(* Logix 5000 project; controller Close_Palletizing 1769-L33ERM rev 33.13; software revision 33.00; part 4 of 5 *)

VAR_GLOBAL   (* controller tags *)
   ActiveUserFrame : DINT := 1;
   ActiveUserFrame_Old : DINT := 1;
   ActiveUserFrame_Timer : TIMER := (PRE := 50, ACC := 21, EN := 1, TT := 1);
   ActiveUserFrameErr : BOOL;
   AirPressure : ALIAS FOR YRC1000_Rbt_Ctlr:I.Data[1].4;   // Sensor on air in, used to verify pressure
   Alarm : ALIAS FOR YRC1000_Rbt_Ctlr:I.Data[8].3;   // Robot in Alarm state
   AlarmReset : ALIAS FOR YRC1000_Rbt_Ctlr:O.Data[0].3;   // Reset alarm output
   AtHomePosition : ALIAS FOR YRC1000_Rbt_Ctlr:I.Data[5].2;
   BatteryAlarm : ALIAS FOR YRC1000_Rbt_Ctlr:I.Data[8].4;   // Robot battery is low
   Blue1 : BOOL;
   Blue2 : BOOL;
   BoltBucketSensor : ALIAS FOR YRC1000_Rbt_Ctlr:I.Data[1].7;   // Sense if the Bolt Bucket is present in the stand
   BothPalletsEmpty : ALIAS FOR Palletizer_full_produced.1;
   BothPalletsFull : ALIAS FOR Palletizer_full_produced.2;
   CallMaster : ALIAS FOR YRC1000_Rbt_Ctlr:O.Data[0].2;   // Call master program to move pointer to top of Master Job
   CallMaster_Timer : TIMER := (PRE := 1000);
   cc_ONS1 : BOOL;
   cc_State : DINT := 100;
   CenterDist : DINT := 303000;
   CheckClearPallet : ALIAS FOR YRC1000_Rbt_Ctlr:I.Data[10].1;
   CheckForComplete : ALIAS FOR YRC1000_Rbt_Ctlr:I.Data[9].5;
   CheckForCompleteAcknowledge : ALIAS FOR YRC1000_Rbt_Ctlr:O.Data[4].6;
   ClearPalletAcknowledge : ALIAS FOR YRC1000_Rbt_Ctlr:O.Data[6].4;
   CloseOffset : DINT := 18;
   Conv_Seq : DINT;
   Conv_Seq_ONS : BOOL := 1;
   ConvConversion2 : REAL := 0.2444492;
   ConveyorActuatorExtend : BOOL;
   ConveyorActuatorRetract : BOOL := 1;
   ConveyorApproachLocation : YRC1000_POSITION_VAR := (Data_Type := 19, Tool_Num := 2, User_Coord_Num := 3, Axis1_Data := -45828, Axis2_Data := 300000, Axis3_Data := 145000, Axis4_Data := 1800000, Axis5_Data := 20000, Axis6_Data := 1800000);
   ConveyorHeight : REAL := 406.29633;   // Distance from UF 3 to the top of the conveyor
   ConveyorPickLocation : YRC1000_POSITION_VAR := (Data_Type := 19, Tool_Num := 2, User_Coord_Num := 3, Axis1_Data := -45828, Axis2_Data := 355000, Axis3_Data := 81500, Axis4_Data := 1800000, Axis5_Data := 20000, Axis6_Data := 1800000);
   ConveyorSequenceReset_Timer : TIMER := (PRE := 3000, ACC := 3000, EN := 1, DN := 1);
   ConveyorSpeed : REAL := 9.301;   // Speed of the conveyor in ft/min
   ConvMul1 : REAL := 1.0;
   ConvMul2 : REAL := 0.99;
   ConvMul3 : REAL := 1.01;
   CurrentPos : REAL[6] := ([0] := 900.002, [1] := 0.001, [2] := 600.006, [3] := -179.9997, [4] := -0.0009, [5] := -0.0009);   // Current position of the active TCP on the robot
   CurrentPos_micro : YRC1000_POSITION_VAR := (Data_Type := 16, Config := 16, Tool_Num := 1, Axis1_Data := 900002, Axis2_Data := 1, Axis3_Data := 600006, Axis4_Data := -1799997, Axis5_Data := -9, Axis6_Data := -9);   // μm
   currentPosErr : BOOL;
   CurrPos_Timer : TIMER := (PRE := 10);
   delay_GoToPick : TIMER := (PRE := 1000);
   delay_LeftPalletOff : TIMER := (PRE := 1000);
   delay_LeftPalletOn : TIMER := (PRE := 1000, ACC := 1000, EN := 1, DN := 1);
   delay_RightPalletOff : TIMER := (PRE := 1000);
   delay_RightPalletOn : TIMER := (PRE := 1000, ACC := 1000, EN := 1, DN := 1);
   DistanceInArray : INT[16] := ([0] := 1976);
        [0]   // Distance sensor reading in MM
   DistanceOutArray : INT[16];
   DistanceSensorValue : DINT := 1978000;
   DoorAccessRequested : ALIAS FOR YRC1000_Rbt_Ctlr:O.Data[5].3;
   DoorLatchRelayPower : ALIAS FOR YRC1000_Rbt_Ctlr:O.Data[2].2;   // Powers the relay that enables the door latch
   DoorRequestAccess : ALIAS FOR YRC1000_Rbt_Ctlr:I.Data[1].0;   // Door Interlock, For request Entry
   DoorUnlocked : ALIAS FOR YRC1000_Rbt_Ctlr:I.Data[2].0;   // The Door Latch is unlocked
   Error_RobotPickupFailed : ALIAS FOR YRC1000_Rbt_Ctlr:I.Data[9].3;
   ExtendedPartWidth : DINT := 693;
   ExtendGripper : ALIAS FOR YRC1000_Rbt_Ctlr:I.Data[9].0;
   ExternalHold : ALIAS FOR YRC1000_Rbt_Ctlr:O.Data[0].1;   // Pauses program execution
   ExternalStart : ALIAS FOR YRC1000_Rbt_Ctlr:O.Data[0].0;   // External command to start the program
   ExtServoOn : ALIAS FOR YRC1000_Rbt_Ctlr:O.Data[0].4;   // External command to turn servos on
   FanucLongPart : DINT := 1072;
   FanucMediumPart : DINT := 795;
   FanucShortPart : DINT := 465;
   GoToPartChange : ALIAS FOR YRC1000_Rbt_Ctlr:O.Data[6].0;
   GoToPick : ALIAS FOR YRC1000_Rbt_Ctlr:O.Data[6].1;
   Green1 : BOOL := 1;
   Green2 : BOOL;
   GrippedPartDistance : DINT := 46000;
   GrippedPartLatchDelay : TIMER := (PRE := 3000);
   HMI_HoldFanuc : BOOL;
   HMI_Manual : BOOL;
   HMI_ParkFanuc : BOOL;
   HMI_Reset : BOOL;
   HMI_Reset_Timer : TIMER := (PRE := 5000);
   HMI_ResetFanuc : BOOL;
   HMI_Start : BOOL;
   HMI_Start_Timer : TIMER := (PRE := 5000);
   HMI_StartFanuc : BOOL;
   HMI_Stop : ALIAS FOR YRC1000_Rbt_Ctlr:O.Data[5].4;
   IFM_Port1_Stroke : Generic_4PORT_IOL := (IOL_Mode := 1, Port_Process_Data_Size := 4, Port_Number := 1, Vendor_ID := 26, Device_ID := 8388785);   // Stroke sensor reading can be found in StrokeInputArray[0]
   IFM_Port2_Distance : Generic_4PORT_IOL := (IOL_Mode := 1, Port_Process_Data_Size := 4, Port_Number := 2, Vendor_ID := 26, Device_ID := 6488065);   // Distance sensor reading can be found in DistanceInArray[0]
   InchesToMove : DINT := 45;
   InHomePosition : ALIAS FOR YRC1000_Rbt_Ctlr:O.Data[5].7;
   InPartChange : ALIAS FOR YRC1000_Rbt_Ctlr:I.Data[9].7;
   InPickApproachAcknowledge : ALIAS FOR YRC1000_Rbt_Ctlr:O.Data[5].2;
   InPlay : ALIAS FOR YRC1000_Rbt_Ctlr:I.Data[8].6;   // Robot is in play mode
   InRemote : ALIAS FOR YRC1000_Rbt_Ctlr:I.Data[8].5;   // Robot is in remote mode
   InTeach : ALIAS FOR YRC1000_Rbt_Ctlr:I.Data[8].7;   // Robot is in teach mode
   LayerNum : DINT := 3;
   LayerPosition : DINT;
   LeftFlashOff : TIMER := (PRE := 750);
   LeftFlashOn : TIMER := (PRE := 750);
   LeftFullRightEmpty : ALIAS FOR Palletizer_full_produced.3;
   LeftIndicator_Green : ALIAS FOR YRC1000_Rbt_Ctlr:O.Data[1].6;   // Indicator light showing the pallet is complete
   LeftIndicator_Yellow : ALIAS FOR YRC1000_Rbt_Ctlr:O.Data[1].7;   // Indicator light showing the pallet is in progress / present
   LeftPalletComplete : ALIAS FOR YRC1000_Rbt_Ctlr:O.Data[4].0;
   LeftPalletPresent : ALIAS FOR YRC1000_Rbt_Ctlr:O.Data[6].6;
   LeftPalletSensor : ALIAS FOR YRC1000_Rbt_Ctlr:I.Data[1].2;   // Sense if a pallet is in the pallet holder
   LeftPalletWillBeNew : BOOL;
   msg_Read_ActiveUserFrame : MESSAGE;
        MessageParameters(ServiceCode := 16#000e, DestinationTag := ActiveUserFrame, ...)
   msg_Read_CurrentPosition : MESSAGE;   // Reading the current position of the robot
        MessageParameters(ServiceCode := 16#0001, DestinationTag := CurrentPos_micro, ...)
   msg_Read_PalletCount : MESSAGE;
        MessageParameters(ServiceCode := 16#000e, DestinationTag := PalletCount, ...)
   msg_Read_PartCount : MESSAGE;   // Reading Part Count from the robot
        MessageParameters(ServiceCode := 16#000e, DestinationTag := PartCount, ...)
   msg_Write_ActiveUserFrame : MESSAGE;
        MessageParameters(ServiceCode := 16#0010, LocalElement := ActiveUserFrame, ...)
   msg_Write_ConveyorApproachLocation : MESSAGE;
        MessageParameters(ServiceCode := 16#0010, LocalElement := ConveyorApproachLocation, ...)
   msg_Write_ConveyorPickLocation : MESSAGE;
        MessageParameters(ServiceCode := 16#0010, LocalElement := ConveyorPickLocation, ...)
   msg_Write_PalletCount : MESSAGE;
        MessageParameters(ServiceCode := 16#0010, LocalElement := PalletCount, ...)
   msg_Write_PalletPlaceLocation : MESSAGE;
        MessageParameters(ServiceCode := 16#0010, LocalElement := RadiatorPlaceLocation, ...)
   msg_Write_PartCount : MESSAGE;
        MessageParameters(ServiceCode := 16#0010, LocalElement := PartCount, ...)
   msg_Write_RadiatorType : MESSAGE;
        MessageParameters(ServiceCode := 16#0010, LocalElement := RadiatorType, ...)
   NewPallet : ALIAS FOR YRC1000_Rbt_Ctlr:O.Data[6].3;
   OffsetDist : DINT := 214000;
   ONS_PartGripped : BOOL;
   ons_SendFanucHome : BOOL;
   ons_StartClearPallet : BOOL;
   PalletCount : DINT := 5;
   PalletCount_old : DINT := 4;
   PalletCount_Timer : TIMER := (PRE := 50, ACC := 9, EN := 1, TT := 1);
   PalletCountErr : BOOL;
   Palletizer_full_produced : DINT := 46596096; {produced}
   PalletNotClear : ALIAS FOR YRC1000_Rbt_Ctlr:O.Data[6].5;
   PalletsNotReady : BOOL;
   PalletStarted : ALIAS FOR YRC1000_Rbt_Ctlr:I.Data[10].2;
   PartCount : DINT := 5;
   PartCount_Timer : TIMER := (PRE := 50, ACC := 10, EN := 1, TT := 1);
   PartCountErr : BOOL;
   PartID_Current : DINT := 7;
   PartInTool : ALIAS FOR YRC1000_Rbt_Ctlr:O.Data[4].2;
   PartLength : DINT := 432;
   PartLength_Current : DINT := 432;   // 17" = 432 mm | 30" = 762 mm | 41" = 1041 mm
   PartMovedOn_Timer : TIMER := (PRE := 14667);
   PartNeverReachedEnd : ALIAS FOR Palletizer_full_produced.6;
   PartNeverReachedEnd_Timer : TIMER := (PRE := 24191);
   PartNum : DINT := 5990261;
   PartNum_Current : DINT := 5990261;
   PartNumber : STRING := '5990261L';
   PartNumber_Current : STRING := '5990261L';
   PartPosition : DINT;
   PartRows : DINT := 3;
   PartRows_Current : DINT := 3;
   PartThickness : REAL := 51.5;
   PartThickness_Current : REAL := 51.5;   // 2r = 34.1-34.6 mm | 3r = 51.1-51.8 mm | 4r = 68.2-68.9 mm
   PartWidth : DINT := 711;
   PartWidth_Current : DINT := 711;   // 14" = 356 mm | 16" = 407 mm | 20" = 508 mm | 22" = 559 mm | 24" = 610 mm | 28" = 711 mm | 32" = 813 mm
   PCConnect : STRING := '1/24/2024 3:13:43 PM';
   Pick_Seq : DINT;
   Pick_Timer : TIMER := (PRE := 1000);
   PickConversion1 : REAL := 3.75;
   PickConversion2 : REAL := 225000.0;
   PickReq_State : DINT := 10;
   PickRequest : ALIAS FOR YRC1000_Rbt_Ctlr:I.Data[9].6;
   PickRequestAcknowledge : ALIAS FOR YRC1000_Rbt_Ctlr:O.Data[5].5;
   PickupConveyorSensor : ALIAS FOR YRC1000_Rbt_Ctlr:I.Data[1].5;   // Sense if the radiator is ready for pickup
   PickupErrorAcknowledge : ALIAS FOR YRC1000_Rbt_Ctlr:O.Data[4].7;
   pickupRecovery : BOOL;
   PickupSensorInactive_Timer : TIMER := (PRE := 5000);
   Place_Error : BOOL;
   PlaceReq_State : DINT := 10;
   PlaceRequestAcknowledge : ALIAS FOR YRC1000_Rbt_Ctlr:O.Data[4].5;
   PN_Timer : TIMER := (PRE := 10);
   Prog_StartFanuc : BOOL;
   QuadStack : ALIAS FOR YRC1000_Rbt_Ctlr:O.Data[5].1;
   RadiatorPicked : ALIAS FOR Palletizer_full_produced.0;
   RadiatorPlaceLocation : YRC1000_POSITION_VAR := (Data_Type := 19, Tool_Num := 8, User_Coord_Num := 1, Axis1_Data := 517000, Axis3_Data := 316750, Axis4_Data := 1800000);
   RadiatorType : DINT := 1;   // 1: 17" 2: 30" 3 41"
   Read_ActiveUserFrame : BOOL;
   Read_CurrPos : BOOL := 1;
   Read_PalletCount : BOOL;
   Read_PartCount : BOOL := 1;
   Release_Timer : TIMER := (PRE := 5000);
   Reset : ALIAS FOR YRC1000_Rbt_Ctlr:I.Data[1].1;   // Door Interlock, For reset Entry
   ResetPalletCount : BOOL;
   RetractGripper : ALIAS FOR YRC1000_Rbt_Ctlr:I.Data[9].1;
   RightFlashOff : TIMER := (PRE := 750, ACC := 174, EN := 1, TT := 1);
   RightFlashOn : TIMER := (PRE := 750, ACC := 750, EN := 1, DN := 1);
   RightFullLeftEmpty : ALIAS FOR Palletizer_full_produced.4;
   RightIndicator_Green : ALIAS FOR YRC1000_Rbt_Ctlr:O.Data[2].0;   // Indicator light showing the pallet is complete
   RightIndicator_Yellow : ALIAS FOR YRC1000_Rbt_Ctlr:O.Data[2].1;   // Indicator light showing the pallet is in progress / present
   RightPalletComplete : ALIAS FOR YRC1000_Rbt_Ctlr:O.Data[4].1;
   RightPalletPresent : ALIAS FOR YRC1000_Rbt_Ctlr:O.Data[6].7;
   RightPalletSensor : ALIAS FOR YRC1000_Rbt_Ctlr:I.Data[1].3;   // Sense if a pallet is in the pallet holder
   RightPalletWillBeNew : BOOL;
   Robot_InPickApproach : ALIAS FOR YRC1000_Rbt_Ctlr:I.Data[9].4;
   RobotCannotPlaceCurrentPart : ALIAS FOR Palletizer_full_produced.5;
   RobotExternalEStop : ALIAS FOR YRC1000_Rbt_Ctlr:I.Data[4].1;
   RobotInsideConveyor : ALIAS FOR YRC1000_Rbt_Ctlr:I.Data[10].0;
   RobotInsideConveyorProduced : ALIAS FOR Palletizer_full_produced.9;
   RobotNotRunning : ALIAS FOR Palletizer_full_produced.7;
   RobotNotSupposedToBeRunning : ALIAS FOR Palletizer_full_produced.8;
   RobotPlaceRequest : ALIAS FOR YRC1000_Rbt_Ctlr:I.Data[9].2;
   RobotTeachPendantEStop : ALIAS FOR YRC1000_Rbt_Ctlr:I.Data[4].2;
   Running : ALIAS FOR YRC1000_Rbt_Ctlr:I.Data[8].0;   // Robot running status
   SafetyCircuitBroken : ALIAS FOR YRC1000_Rbt_Ctlr:I.Data[4].0;
   SafetyRelayReset : ALIAS FOR YRC1000_Rbt_Ctlr:O.Data[2].3;   // Reset the safety relays linked to the Pilz sensors
   SecondConveyorSensor : ALIAS FOR YRC1000_Rbt_Ctlr:I.Data[1].6;   // Sense if a coil is waiting on the conveyor
   SelectPlay : ALIAS FOR YRC1000_Rbt_Ctlr:O.Data[0].5;   // External command to put robot in play mode
   SelectTeach : ALIAS FOR YRC1000_Rbt_Ctlr:O.Data[0].6;   // External command to put robot in teach mode
   ServoOn : ALIAS FOR YRC1000_Rbt_Ctlr:I.Data[8].1;   // Servo on status
   SideDist : DINT;
   SingleStack : ALIAS FOR YRC1000_Rbt_Ctlr:O.Data[5].0;
   StackLight_Blue : ALIAS FOR YRC1000_Rbt_Ctlr:O.Data[1].3;   // Blue on the light stack
   StackLight_Buzzer : ALIAS FOR YRC1000_Rbt_Ctlr:O.Data[1].0;   // Buzzer on the stack light
   StackLight_Green : ALIAS FOR YRC1000_Rbt_Ctlr:O.Data[1].5;   // Green light on light stack
   StackLight_Red : ALIAS FOR YRC1000_Rbt_Ctlr:O.Data[1].2;   // Red light on light stack
   StackLight_White : ALIAS FOR YRC1000_Rbt_Ctlr:O.Data[1].1;   // White on the light stack
   StackLight_Yellow : ALIAS FOR YRC1000_Rbt_Ctlr:O.Data[1].4;   // Yellow light on light stack
   state_CheckClearPallet : DINT := 100;
   StillOnOldPart_Timer : TIMER := (PRE := 500);
   StrokeInputArray : INT[16] := ([0] := 13136);
   StrokeOutputArray : INT[16];
   StrokePosition : DINT := 821;   // Gripper Cylinder position GTE 700 = Retracted LTE 100 = Extended
   test_bit_1 : BOOL := 1;
   test_bit_2 : BOOL;
   test_bit_3 : BOOL := 1;
   test_toggle : BOOL;
   ThirdConveyorSensor : BOOL;
   timer_FanucReset : TIMER := (PRE := 500);
   timer_FanucStart : TIMER := (PRE := 500);
   timer_GreenFlashOff : TIMER := (PRE := 1000, ACC := 1000, EN := 1, DN := 1);
   timer_GreenFlashOn : TIMER := (PRE := 1000, ACC := 351, EN := 1, TT := 1);
   ToolExtended : ALIAS FOR YRC1000_Rbt_Ctlr:O.Data[4].3;
   ToolRetracted : ALIAS FOR YRC1000_Rbt_Ctlr:O.Data[4].4;
   ToPC_AirPressure : DINT := 1;
   ToPC_BoltBucketSensor : DINT := 1;
   ToPC_ConveyorStatus : DINT;
   ToPC_DoorStatus : DINT;
   ToPC_FanucFault : DINT := 1;
   ToPC_FanucRunning : DINT;
   ToPC_LeftPalletStatus : DINT := 1;
   ToPC_PalletNotClear : DINT;
   ToPC_PickupFailed : DINT;
   ToPC_PlaceError : DINT;
   ToPC_RightPalletStatus : DINT := 2;
   ToPC_RobotEStop : DINT;
   ToPC_RobotRunning : DINT := 1;
   ToPC_SafetyCircuitBroken : DINT;
   ToPC_ToolStatus : DINT;
   TopOfMaster : ALIAS FOR YRC1000_Rbt_Ctlr:I.Data[8].2;   // Top of Master Job
   TurnOffBuzzer : BOOL;
   TwoStack : ALIAS FOR YRC1000_Rbt_Ctlr:O.Data[6].2;
   WaitingForPartAtEnd : BOOL;
   Write_ActiveUserFrame : BOOL;
   Write_ActiveUserFrame1 : BOOL;
   Write_ConveyorLocations : BOOL;
   Write_PalletPlaceLocation : BOOL;
   Write_PartCount : BOOL;
   Write_RadiatorType : BOOL;
END_VAR

PROGRAM MainProgram   (* main routine MainRoutine *)
VAR
   ActuatorCloseTime : REAL := 0.75;
   ConvConversion : REAL := 74.50812;
   ConvConversion1 : REAL := 6.2090096;
   ConveyorLocations_ONS : BOOL;
   ConvMultiplier : REAL := 1.0;
   ToggleStokeAOI : BOOL := 1;
   Write_ActiveUserFrame2 : BOOL;
END_VAR

ROUTINE Fanuc_Communication   (* ladder *)
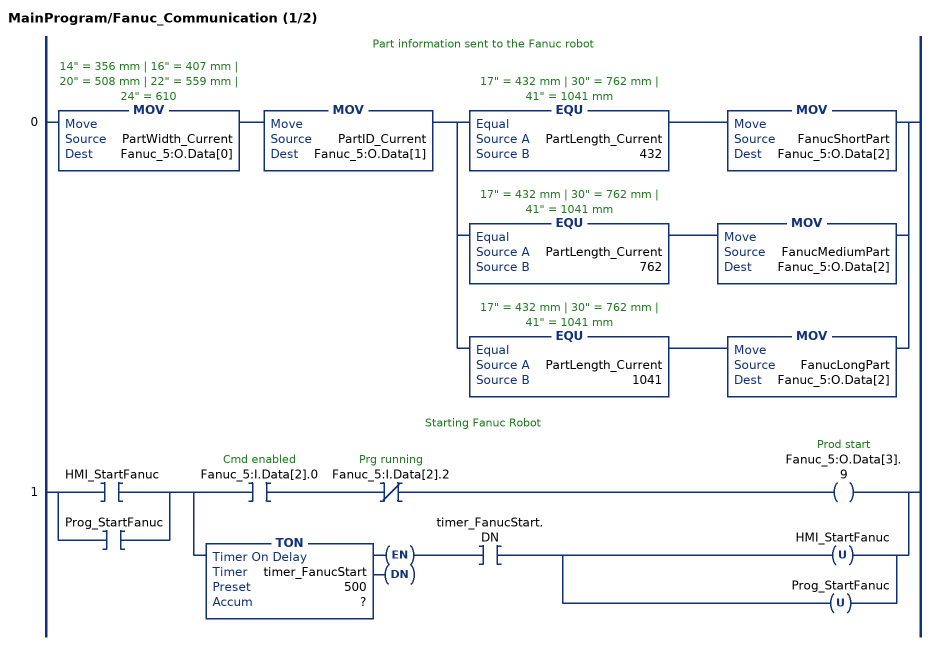
   // Part information sent to the Fanuc robot
   0: MOV(PartWidth_Current,Fanuc_5:O.Data[0])MOV(PartID_Current,Fanuc_5:O.Data[1])[EQU(PartLength_Current,432) MOV(FanucShortPart,Fanuc_5:O.Data[2]) ,EQU(PartLength_Current,762) MOV(FanucMediumPart,Fanuc_5:O.Data[2]) ,EQU(PartLength_Current,1041) MOV(FanucLongPart,Fanuc_5:O.Data[2]) ];
   // Starting Fanuc Robot
   1: [XIC(HMI_StartFanuc) ,XIC(Prog_StartFanuc) ][XIC(Fanuc_5:I.Data[2].0) XIO(Fanuc_5:I.Data[2].2) OTE(Fanuc_5:O.Data[3].9) ,TON(timer_FanucStart,?,?) XIC(timer_FanucStart.DN) [OTU(HMI_StartFanuc) ,OTU(Prog_StartFanuc) ] ];
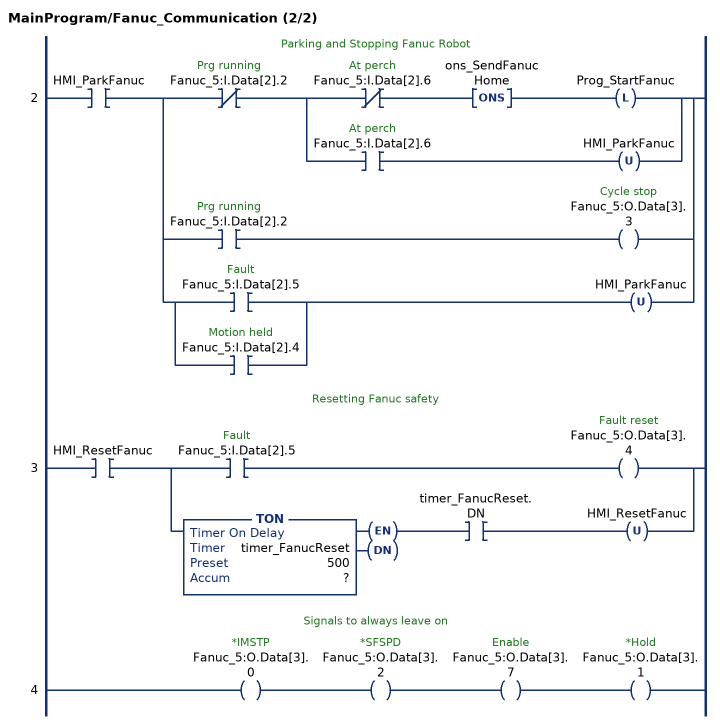
   // Parking and Stopping Fanuc Robot
   2: XIC(HMI_ParkFanuc)[[XIO(Fanuc_5:I.Data[2].2) [XIO(Fanuc_5:I.Data[2].6) ONS(ons_SendFanucHome) OTL(Prog_StartFanuc) ,XIC(Fanuc_5:I.Data[2].6) OTU(HMI_ParkFanuc) ] ,XIC(Fanuc_5:I.Data[2].2) OTE(Fanuc_5:O.Data[3].3) ] ,[XIC(Fanuc_5:I.Data[2].5) ,XIC(Fanuc_5:I.Data[2].4) ] OTU(HMI_ParkFanuc) ];
   // Resetting Fanuc safety
   3: XIC(HMI_ResetFanuc)[XIC(Fanuc_5:I.Data[2].5) OTE(Fanuc_5:O.Data[3].4) ,TON(timer_FanucReset,?,?) XIC(timer_FanucReset.DN) OTU(HMI_ResetFanuc) ];
   // Signals to always leave on
   4: OTE(Fanuc_5:O.Data[3].0)OTE(Fanuc_5:O.Data[3].2)OTE(Fanuc_5:O.Data[3].7)OTE(Fanuc_5:O.Data[3].1);
END_ROUTINE

ROUTINE Fanuc_PartID   (* structured text *)
   if PartLength_Current = 432 then
   	if PartWidth_Current = 356 then
   		PartID_Current := 1;
   	elsif PartWidth_Current = 406 then
   		PartID_Current := 2;
   	elsif PartWidth_Current = 508 then
   		if PartRows_Current = 2 then
   			PartID_Current := 3;
   		elsif PartRows_Current = 3 then
   			PartID_Current := 4;
   		end_if;
   	elsif PartWidth_Current = 559 then
   		PartID_Current := 5;
   	elsif PartWidth_Current = 610 then
   		PartID_Current := 6;
   	elsif PartWidth_Current = 711 then
   		if PartRows_Current = 3 then
   			PartID_Current := 7;
   		elsif PartRows_Current = 4 then
   			PartID_Current := 8;
   		end_if;
   	elsif PartWidth_Current = 813 then
   		PartID_Current := 9;
   	end_if;
   elsif PartLength_Current = 762 then
   	if PartRows_Current = 2 then
   		PartID_Current := 10;
   	elsif PartRows_Current = 3 then
   		PartID_Current := 11;
   	end_if;
   elsif PartLength_Current = 1041 then
   	if PartRows_Current = 3 then
   		PartID_Current := 12;
   	elsif PartRows_Current = 4 then
   		PartID_Current := 13;
   	end_if;
   end_if;
END_ROUTINE

ROUTINE IO_Link   (* ladder *)
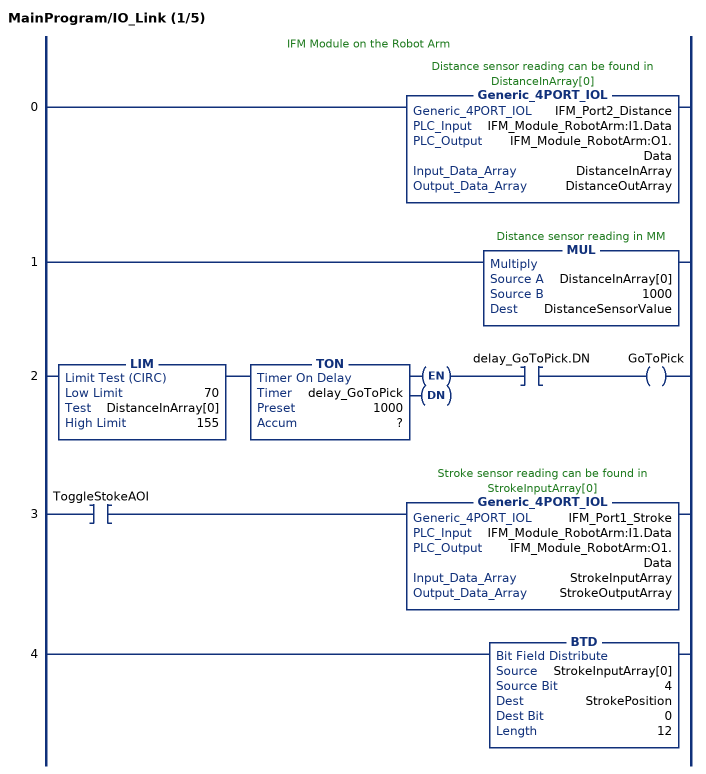
   // IFM Module on the Robot Arm
   0: Generic_4PORT_IOL(IFM_Port2_Distance,IFM_Module_RobotArm:I1.Data,IFM_Module_RobotArm:O1.Data,DistanceInArray,DistanceOutArray);
   1: MUL(DistanceInArray[0],1000,DistanceSensorValue);
   2: LIM(70,DistanceInArray[0],155)TON(delay_GoToPick,?,?)XIC(delay_GoToPick.DN)OTE(GoToPick);
   3: XIC(ToggleStokeAOI)Generic_4PORT_IOL(IFM_Port1_Stroke,IFM_Module_RobotArm:I1.Data,IFM_Module_RobotArm:O1.Data,StrokeInputArray,StrokeOutputArray);
   4: BTD(StrokeInputArray[0],4,StrokePosition,0,12);
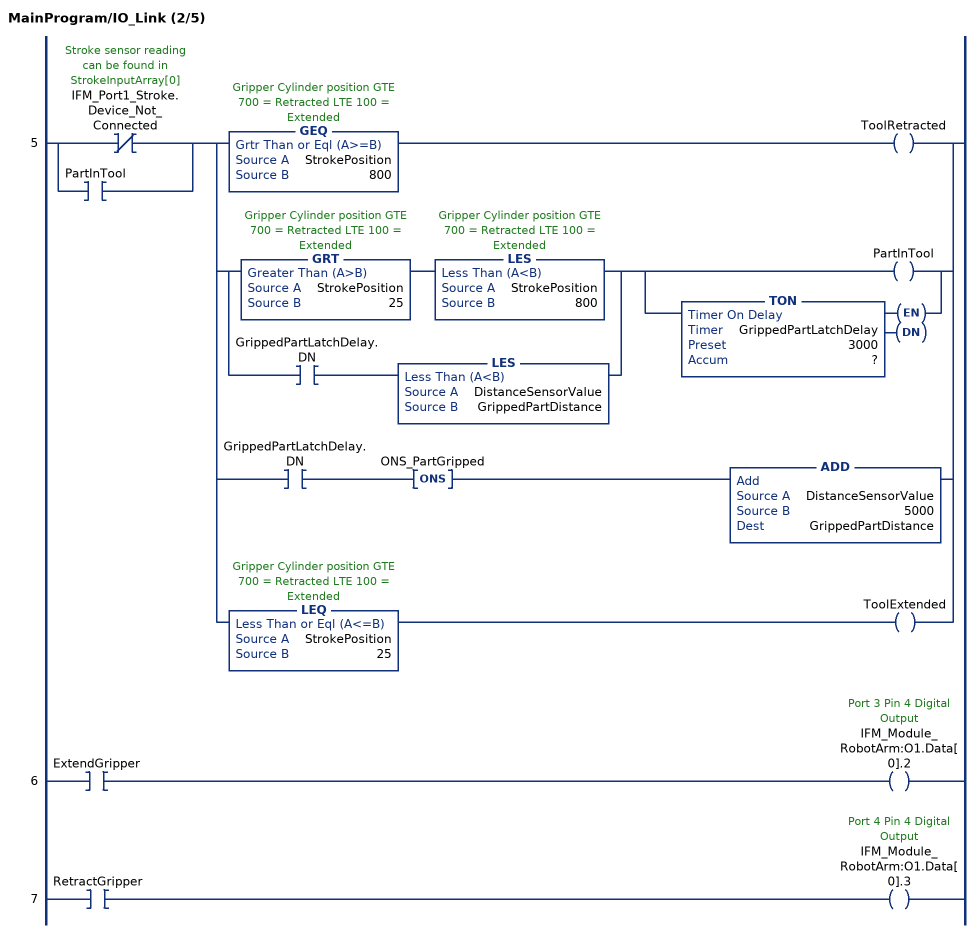
   5: [XIO(IFM_Port1_Stroke.Device_Not_Connected) ,XIC(PartInTool) ][GEQ(StrokePosition,800) OTE(ToolRetracted) ,[GRT(StrokePosition,25) LES(StrokePosition,800) ,XIC(GrippedPartLatchDelay.DN) LES(DistanceSensorValue,GrippedPartDistance) ] [OTE(PartInTool) ,TON(GrippedPartLatchDelay,?,?) ] ,XIC(GrippedPartLatchDelay.DN) ONS(ONS_PartGripped) ADD(DistanceSensorValue,5000,GrippedPartDistance) ,LEQ(StrokePosition,25) OTE(ToolExtended) ];
   6: XIC(ExtendGripper)OTE(IFM_Module_RobotArm:O1.Data[0].2);
   7: XIC(RetractGripper)OTE(IFM_Module_RobotArm:O1.Data[0].3);
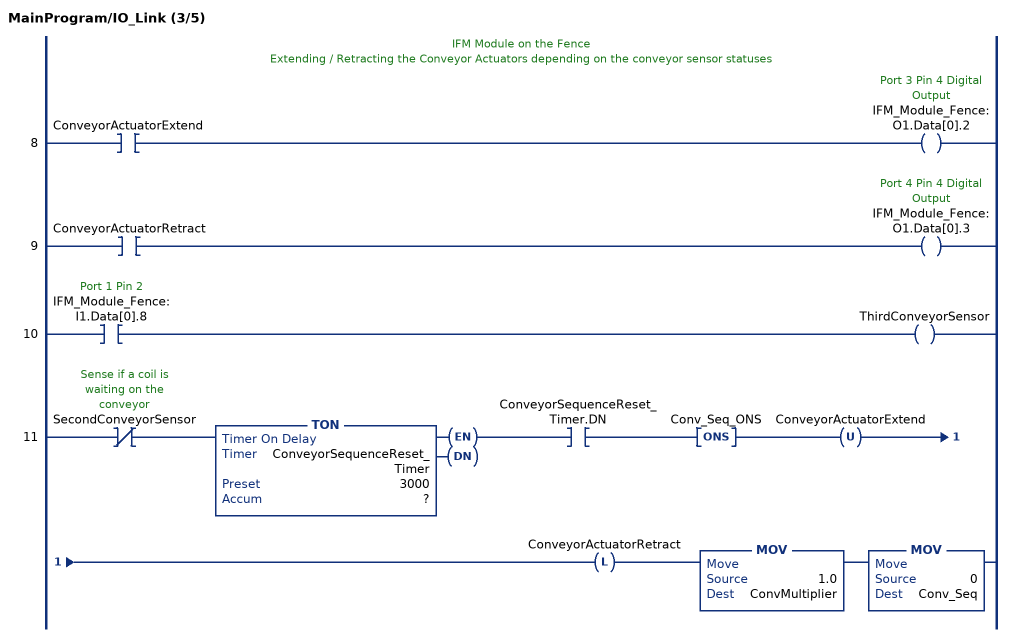
   // IFM Module on the Fence
   // Extending / Retracting the Conveyor Actuators depending on the conveyor sensor statuses
   8: XIC(ConveyorActuatorExtend)OTE(IFM_Module_Fence:O1.Data[0].2);
   9: XIC(ConveyorActuatorRetract)OTE(IFM_Module_Fence:O1.Data[0].3);
   10: XIC(IFM_Module_Fence:I1.Data[0].8)OTE(ThirdConveyorSensor);
   11: XIO(SecondConveyorSensor)TON(ConveyorSequenceReset_Timer,?,?)XIC(ConveyorSequenceReset_Timer.DN)ONS(Conv_Seq_ONS)OTU(ConveyorActuatorExtend)OTL(ConveyorActuatorRetract)MOV(1.0,ConvMultiplier)MOV(0,Conv_Seq);
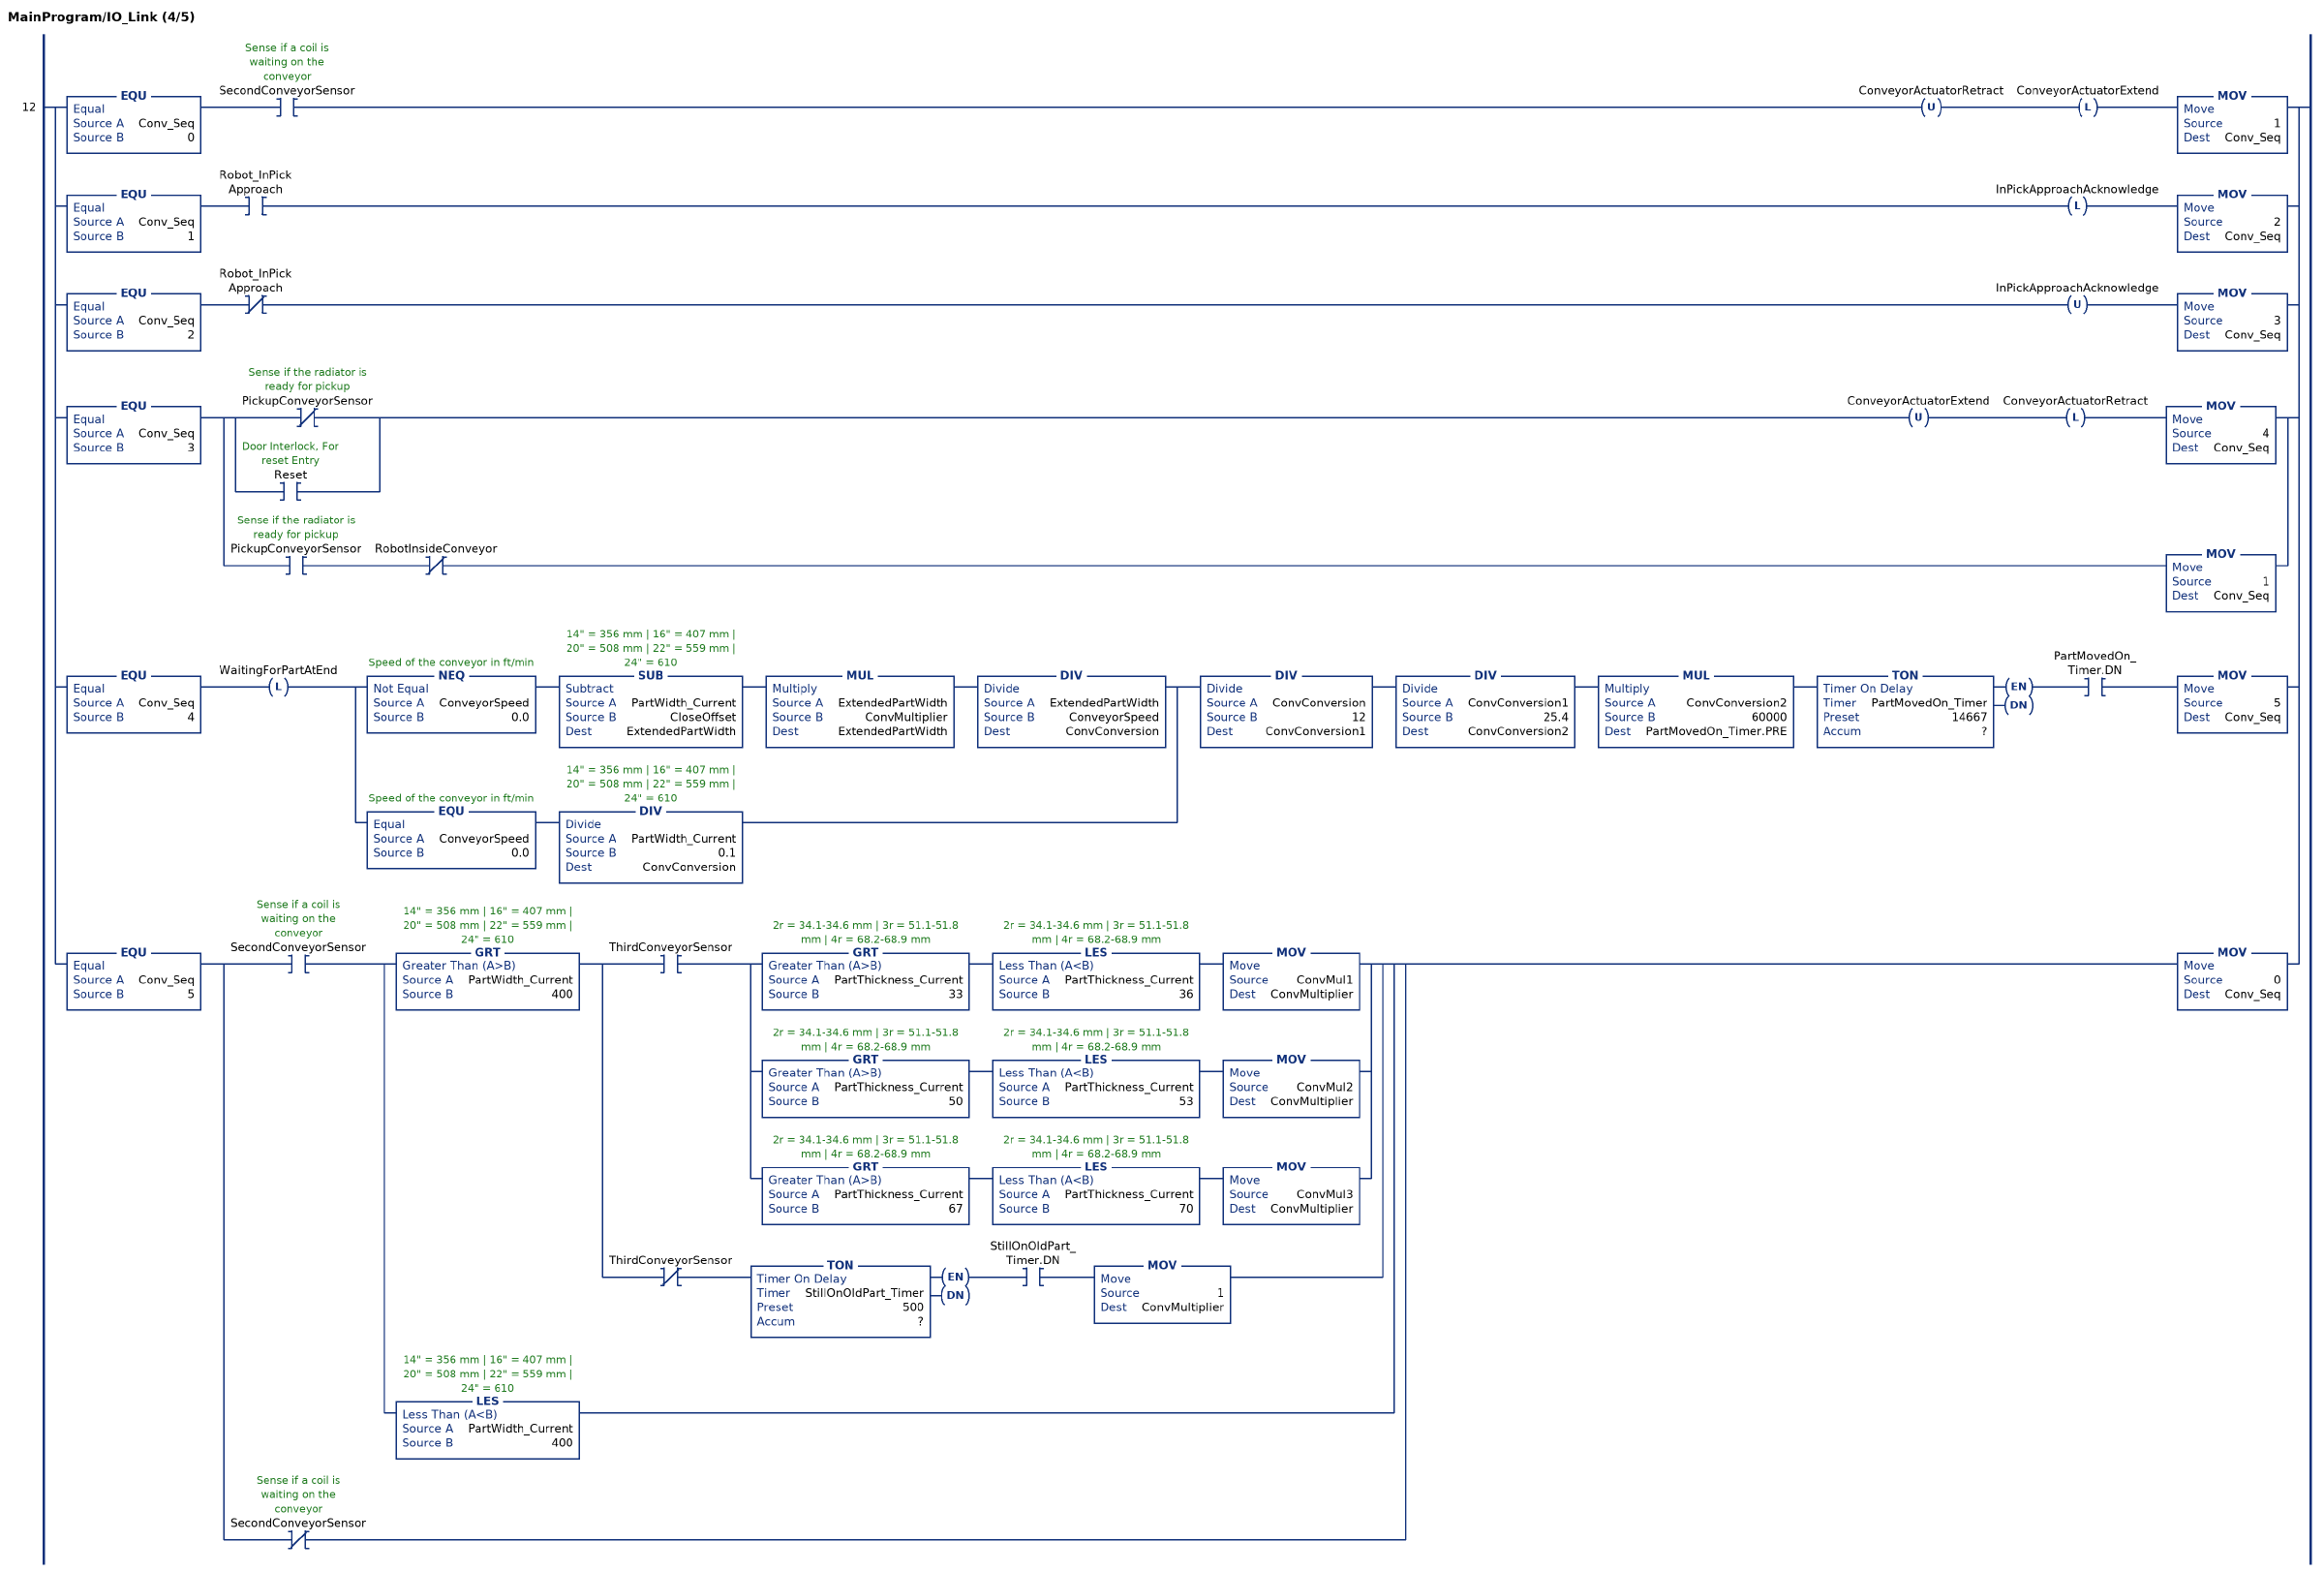
   12: [EQU(Conv_Seq,0) XIC(SecondConveyorSensor) OTU(ConveyorActuatorRetract) OTL(ConveyorActuatorExtend) MOV(1,Conv_Seq) ,EQU(Conv_Seq,1) XIC(Robot_InPickApproach) OTL(InPickApproachAcknowledge) MOV(2,Conv_Seq) ,EQU(Conv_Seq,2) XIO(Robot_InPickApproach) OTU(InPickApproachAcknowledge) MOV(3,Conv_Seq) ,EQU(Conv_Seq,3) [[XIO(PickupConveyorSensor) ,XIC(Reset) ] OTU(ConveyorActuatorExtend) OTL(ConveyorActuatorRetract) MOV(4,Conv_Seq) ,XIC(PickupConveyorSensor) XIO(RobotInsideConveyor) MOV(1,Conv_Seq) ] ,EQU(Conv_Seq,4) OTL(WaitingForPartAtEnd) [NEQ(ConveyorSpeed,0.0) SUB(PartWidth_Current,CloseOffset,ExtendedPartWidth) MUL(ExtendedPartWidth,ConvMultiplier,ExtendedPartWidth) DIV(ExtendedPartWidth,ConveyorSpeed,ConvConversion) ,EQU(ConveyorSpeed,0.0) DIV(PartWidth_Current,0.1,ConvConversion) ] DIV(ConvConversion,12,ConvConversion1) DIV(ConvConversion1,25.4,ConvConversion2) MUL(ConvConversion2,60000,PartMovedOn_Timer.PRE) TON(PartMovedOn_Timer,?,?) XIC(PartMovedOn_Timer.DN) MOV(5,Conv_Seq) ,EQU(Conv_Seq,5) [XIC(SecondConveyorSensor) [GRT(PartWidth_Current,400) [XIC(ThirdConveyorSensor) [GRT(PartThickness_Current,33) LES(PartThickness_Current,36) MOV(ConvMul1,ConvMultiplier) ,GRT(PartThickness_Current,50) LES(PartThickness_Current,53) MOV(ConvMul2,ConvMultiplier) ,GRT(PartThickness_Current,67) LES(PartThickness_Current,70) MOV(ConvMul3,ConvMultiplier) ] ,XIO(ThirdConveyorSensor) TON(StillOnOldPart_Timer,?,?) XIC(StillOnOldPart_Timer.DN) MOV(1,ConvMultiplier) ] ,LES(PartWidth_Current,400) ] ,XIO(SecondConveyorSensor) ] MOV(0,Conv_Seq) ];
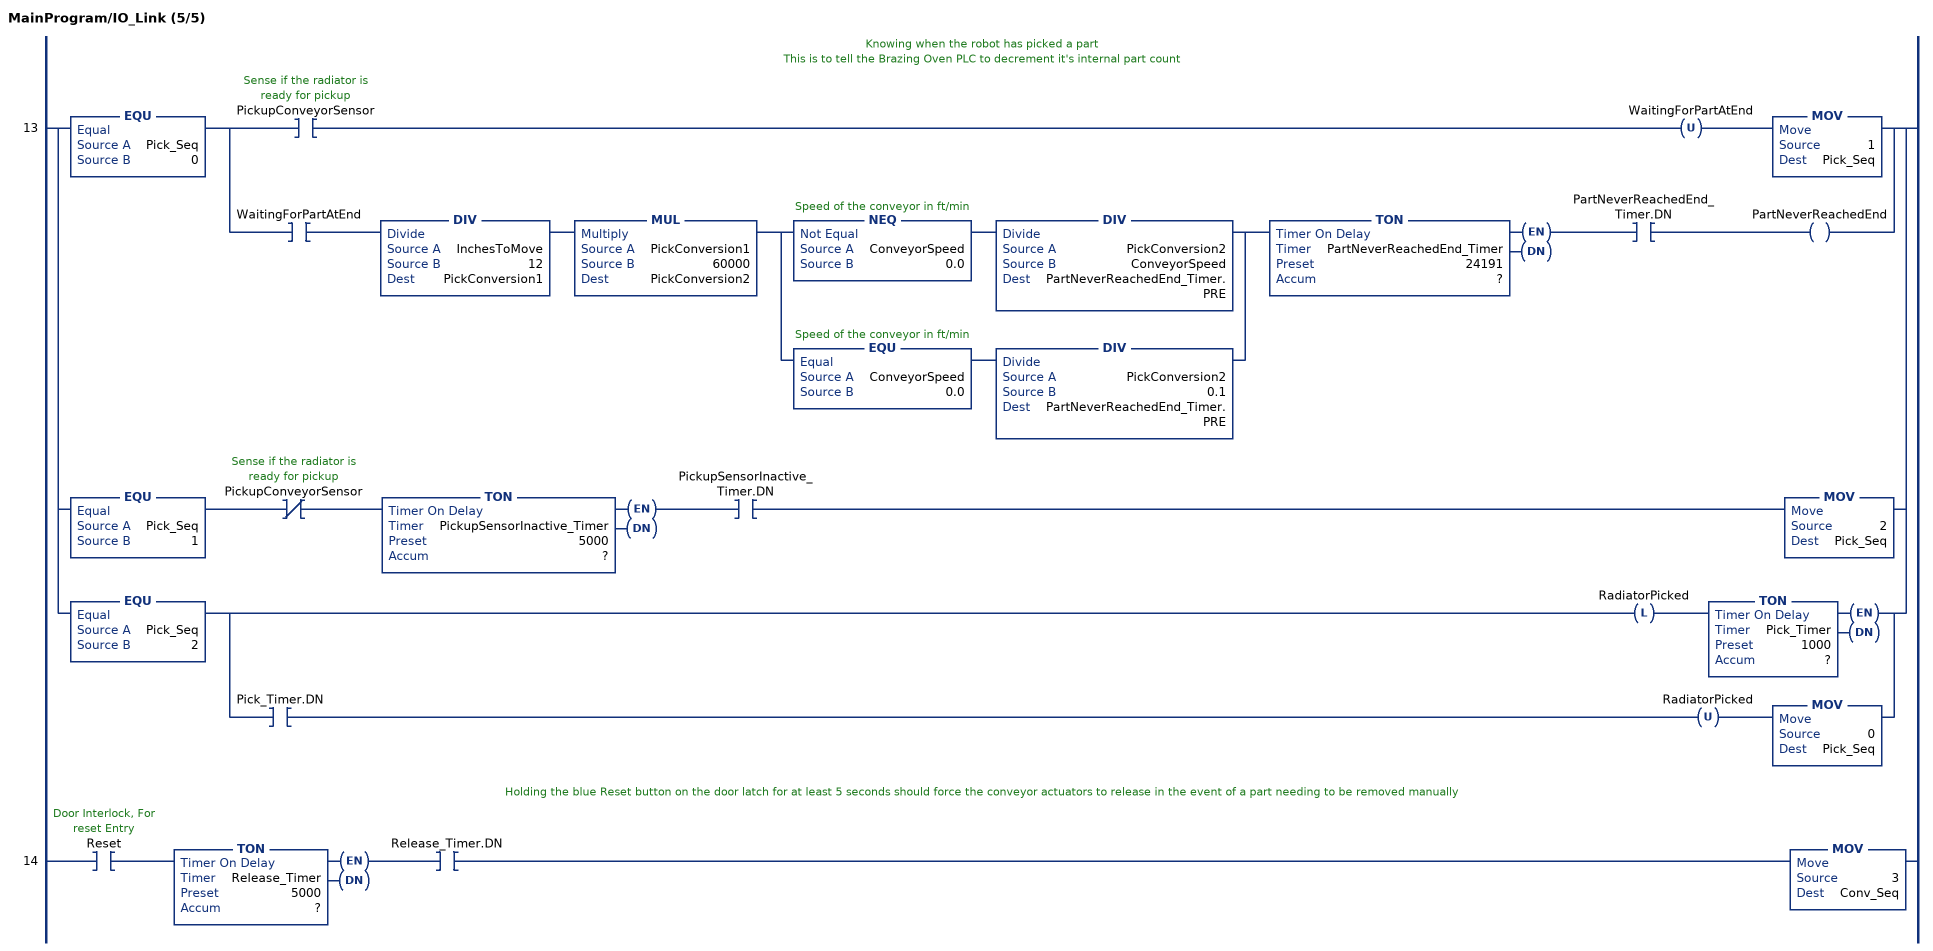
   // Knowing when the robot has picked a part
   // This is to tell the Brazing Oven PLC to decrement it's internal part count
   13: [EQU(Pick_Seq,0) [XIC(PickupConveyorSensor) OTU(WaitingForPartAtEnd) MOV(1,Pick_Seq) ,XIC(WaitingForPartAtEnd) DIV(InchesToMove,12,PickConversion1) MUL(PickConversion1,60000,PickConversion2) [NEQ(ConveyorSpeed,0.0) DIV(PickConversion2,ConveyorSpeed,PartNeverReachedEnd_Timer.PRE) ,EQU(ConveyorSpeed,0.0) DIV(PickConversion2,0.1,PartNeverReachedEnd_Timer.PRE) ] TON(PartNeverReachedEnd_Timer,?,?) XIC(PartNeverReachedEnd_Timer.DN) OTE(PartNeverReachedEnd) ] ,EQU(Pick_Seq,1) XIO(PickupConveyorSensor) TON(PickupSensorInactive_Timer,?,?) XIC(PickupSensorInactive_Timer.DN) MOV(2,Pick_Seq) ,EQU(Pick_Seq,2) [OTL(RadiatorPicked) TON(Pick_Timer,?,?) ,XIC(Pick_Timer.DN) OTU(RadiatorPicked) MOV(0,Pick_Seq) ] ];
   // Holding the blue Reset button on the door latch for at least 5 seconds should force the conveyor actuators to release in the event of a part needing to be removed manually
   14: XIC(Reset)TON(Release_Timer,?,?)XIC(Release_Timer.DN)MOV(3,Conv_Seq);
END_ROUTINE

ROUTINE MainRoutine   (* ladder *)
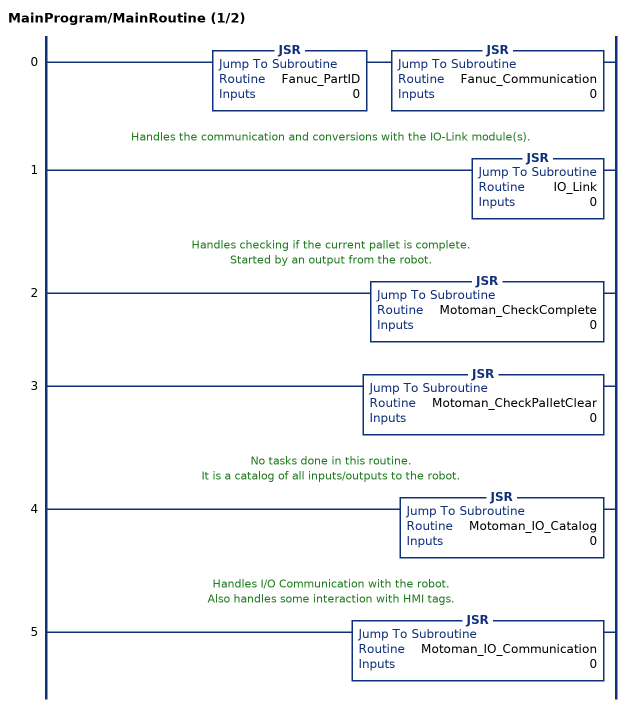
   0: JSR(Fanuc_PartID,0)JSR(Fanuc_Communication,0);
   // Handles the communication and conversions with the IO-Link module(s).
   1: JSR(IO_Link,0);
   // Handles checking if the current pallet is complete.
   // Started by an output from the robot.
   2: JSR(Motoman_CheckComplete,0);
   3: JSR(Motoman_CheckPalletClear,0);
   // No tasks done in this routine.
   // It is a catalog of all inputs/outputs to the robot.
   4: JSR(Motoman_IO_Catalog,0);
   // Handles I/O Communication with the robot.
   // Also handles some interaction with HMI tags.
   5: JSR(Motoman_IO_Communication,0);
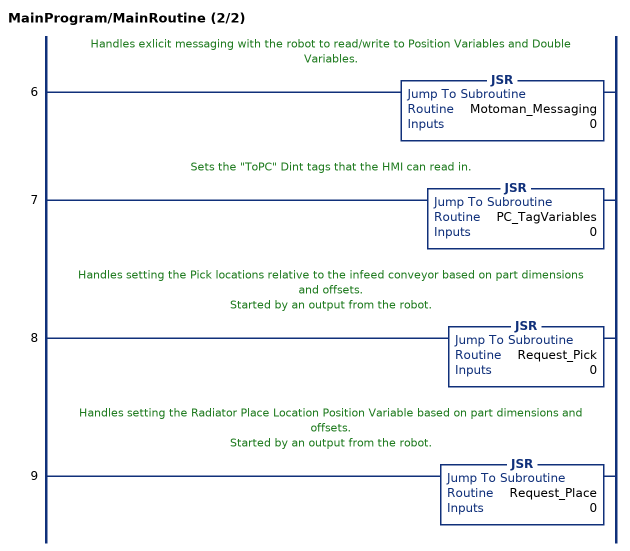
   // Handles exlicit messaging with the robot to read/write to Position Variables and Double Variables.
   6: JSR(Motoman_Messaging,0);
   // Sets the "ToPC" Dint tags that the HMI can read in.
   7: JSR(PC_TagVariables,0);
   // Handles setting the Pick locations relative to the infeed conveyor based on part dimensions and offsets.
   // Started by an output from the robot.
   8: JSR(Request_Pick,0);
   // Handles setting the Radiator Place Location Position Variable based on part dimensions and offsets.
   // Started by an output from the robot.
   9: JSR(Request_Place,0);
END_ROUTINE

ROUTINE Motoman_CheckComplete   (* ladder *)
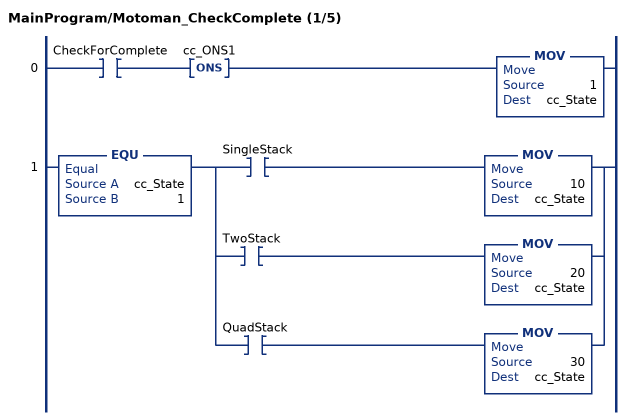
   0: XIC(CheckForComplete)ONS(cc_ONS1)MOV(1,cc_State);
   1: EQU(cc_State,1)[XIC(SingleStack) MOV(10,cc_State) ,XIC(TwoStack) MOV(20,cc_State) ,XIC(QuadStack) MOV(30,cc_State) ];
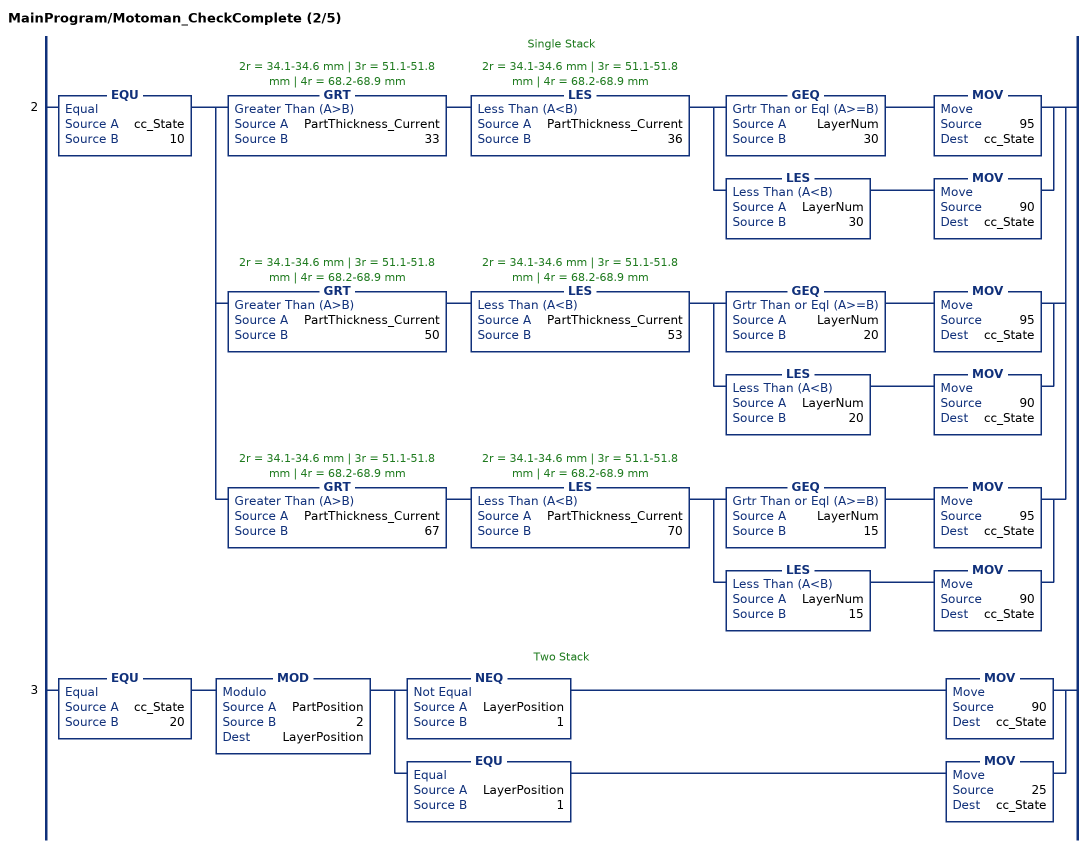
   // Single Stack
   2: EQU(cc_State,10)[GRT(PartThickness_Current,33) LES(PartThickness_Current,36) [GEQ(LayerNum,30) MOV(95,cc_State) ,LES(LayerNum,30) MOV(90,cc_State) ] ,GRT(PartThickness_Current,50) LES(PartThickness_Current,53) [GEQ(LayerNum,20) MOV(95,cc_State) ,LES(LayerNum,20) MOV(90,cc_State) ] ,GRT(PartThickness_Current,67) LES(PartThickness_Current,70) [GEQ(LayerNum,15) MOV(95,cc_State) ,LES(LayerNum,15) MOV(90,cc_State) ] ];
   // Two Stack
   3: EQU(cc_State,20)MOD(PartPosition,2,LayerPosition)[NEQ(LayerPosition,1) MOV(90,cc_State) ,EQU(LayerPosition,1) MOV(25,cc_State) ];
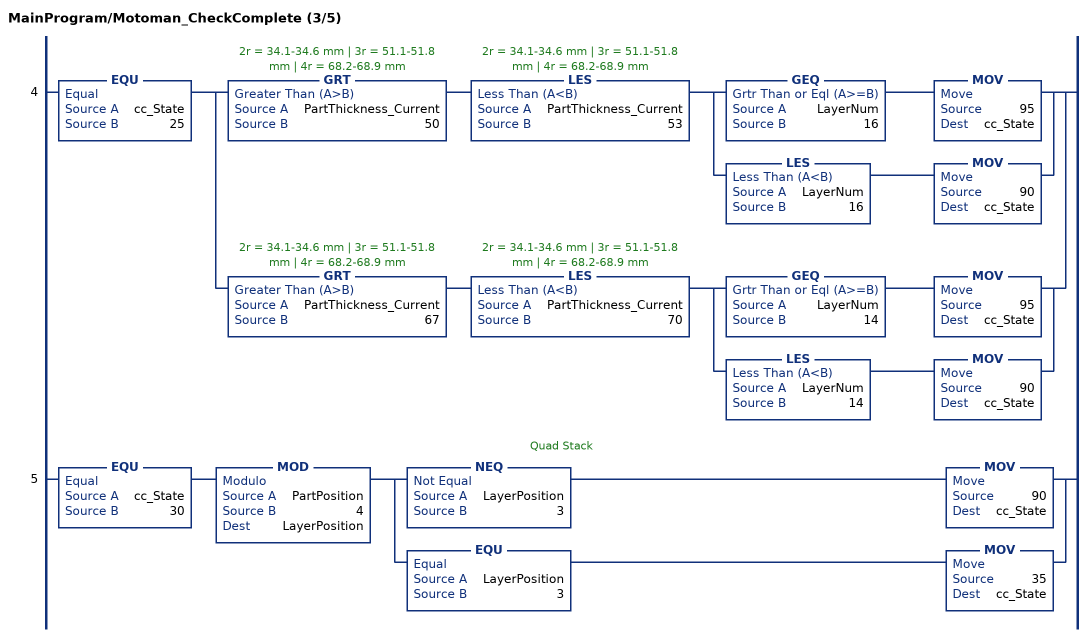
   4: EQU(cc_State,25)[GRT(PartThickness_Current,50) LES(PartThickness_Current,53) [GEQ(LayerNum,16) MOV(95,cc_State) ,LES(LayerNum,16) MOV(90,cc_State) ] ,GRT(PartThickness_Current,67) LES(PartThickness_Current,70) [GEQ(LayerNum,14) MOV(95,cc_State) ,LES(LayerNum,14) MOV(90,cc_State) ] ];
   // Quad Stack
   5: EQU(cc_State,30)MOD(PartPosition,4,LayerPosition)[NEQ(LayerPosition,3) MOV(90,cc_State) ,EQU(LayerPosition,3) MOV(35,cc_State) ];
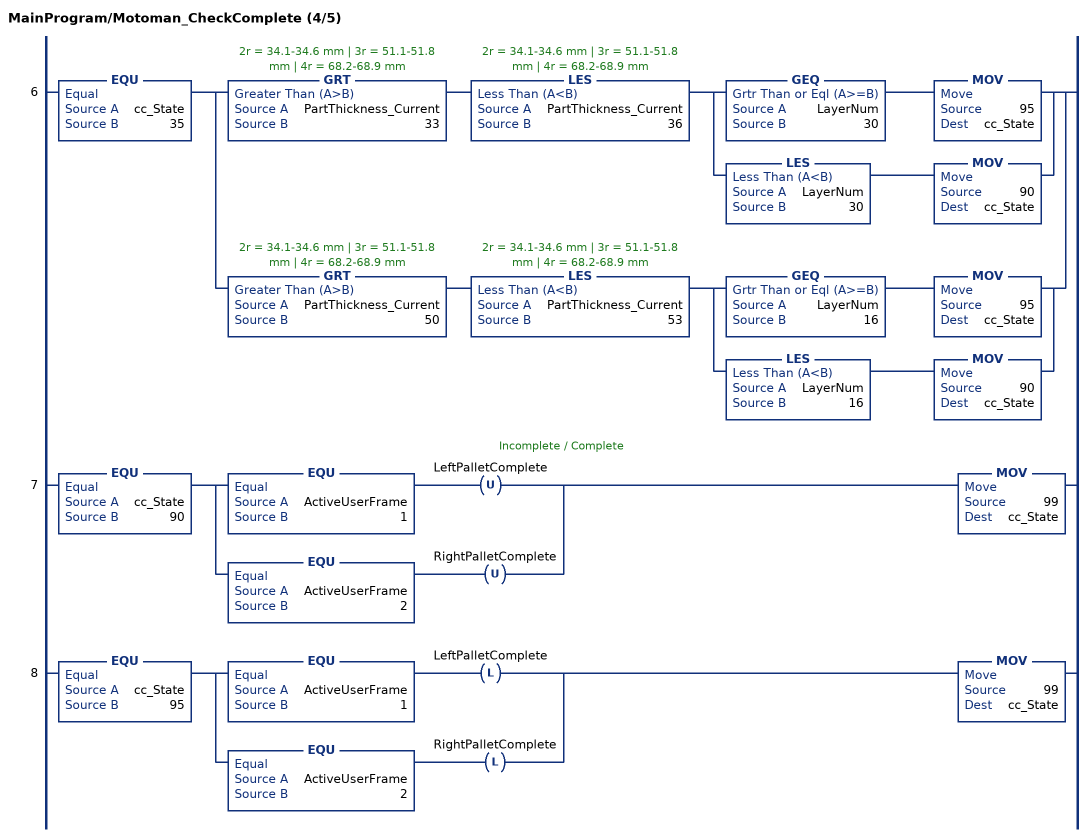
   6: EQU(cc_State,35)[GRT(PartThickness_Current,33) LES(PartThickness_Current,36) [GEQ(LayerNum,30) MOV(95,cc_State) ,LES(LayerNum,30) MOV(90,cc_State) ] ,GRT(PartThickness_Current,50) LES(PartThickness_Current,53) [GEQ(LayerNum,16) MOV(95,cc_State) ,LES(LayerNum,16) MOV(90,cc_State) ] ];
   // Incomplete / Complete
   7: EQU(cc_State,90)[EQU(ActiveUserFrame,1) OTU(LeftPalletComplete) ,EQU(ActiveUserFrame,2) OTU(RightPalletComplete) ]MOV(99,cc_State);
   8: EQU(cc_State,95)[EQU(ActiveUserFrame,1) OTL(LeftPalletComplete) ,EQU(ActiveUserFrame,2) OTL(RightPalletComplete) ]MOV(99,cc_State);
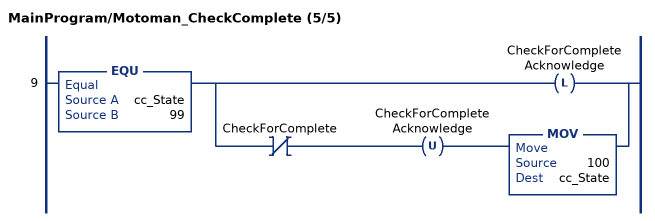
   9: EQU(cc_State,99)[OTL(CheckForCompleteAcknowledge) ,XIO(CheckForComplete) OTU(CheckForCompleteAcknowledge) MOV(100,cc_State) ];
END_ROUTINE

ROUTINE Motoman_CheckPalletClear   (* ladder *)
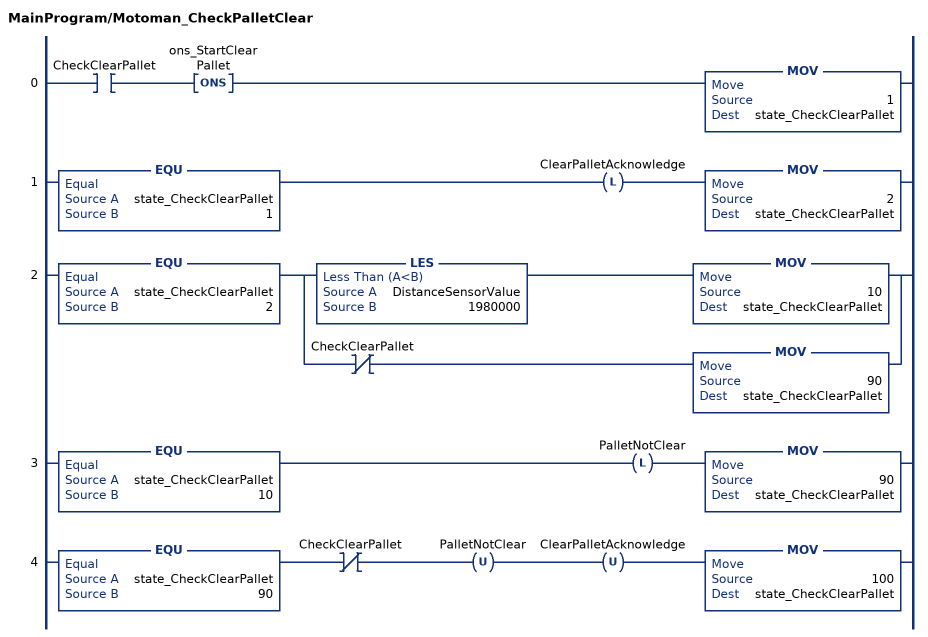
   0: XIC(CheckClearPallet)ONS(ons_StartClearPallet)MOV(1,state_CheckClearPallet);
   1: EQU(state_CheckClearPallet,1)OTL(ClearPalletAcknowledge)MOV(2,state_CheckClearPallet);
   2: EQU(state_CheckClearPallet,2)[LES(DistanceSensorValue,1980000) MOV(10,state_CheckClearPallet) ,XIO(CheckClearPallet) MOV(90,state_CheckClearPallet) ];
   3: EQU(state_CheckClearPallet,10)OTL(PalletNotClear)MOV(90,state_CheckClearPallet);
   4: EQU(state_CheckClearPallet,90)XIO(CheckClearPallet)OTU(PalletNotClear)OTU(ClearPalletAcknowledge)MOV(100,state_CheckClearPallet);
END_ROUTINE

ROUTINE Motoman_IO_Catalog   (* ladder *)
   // Physical Inputs
   //  These signals come directly from sensors/devices and get passed from the Robot to the PLC
   //  Name                       Robot Input     Ext. Input Signal     Ext. Output Signal     PLC Input
   // --------------------------------------------------------------------------------------------------
   //  Entry Request                IN 001             20030                 30080            I.Data[1].0
   //  Safety Relay Reset           IN 002             20031                 30081            I.Data[1].1
   //  Left Pallet Present          IN 003             20032                 30082            I.Data[1].2
   //  Right Pallet Present         IN 004             20033                 30083            I.Data[4].3
   //  Air Pressure                 IN 005             20034                 30084            I.Data[1].4
   //  Pickup Conveyor Sensor       IN 006             20035                 30085            I.Data[1].5
   //  Backup Conveyor Sensor       IN 007             20036                 30086            I.Data[1].6
   //  Bolt Bucket Sensor           IN 008             20037                 30087            I.Data[1].7
   //  Door Unlocked                IN 009             20040                 30090            I.Data[2].0
   0: NOP();
   // Physical Outputs
   //  These signals are controlled by the PLC. Virtual signals are sent from the PLC to the Robot to know which physical outputs to power.
   //  Name                     Robot Input     Ext. Input Signal     Ext. Output Signal     PLC Output
   // ---------------------------------------------------------------------------------------------------
   //  Stack Light Buzzer         IN 041          20080 / 00060            30030             O.Data[1].0
   //  Stack Light White          IN 042          20081 / 00060            30031             O.Data[1].1
   //  Stack Light Red            IN 043          20082 / 00062            30032             O.Data[1].2
   //  Stack Light Blue           IN 044          20083 / 00063            30033             O.Data[1].3
   //  Stack Light Yellow         IN 045          20084 / 00064            30034             O.Data[1].4
   //  Stack Light Green          IN 046          20085 / 00065            30035             O.Data[1].5
   //  Left Indicator Green       IN 047          20086 / 00066            30036             O.Data[1].6
   //  Left Indicator Yellow      IN 048          20087 / 00067            30037             O.Data[1].7
   //  Right Indicator Green      IN 049          20090 / 00070            30040             O.Data[2].0
   //  Right Indicator Yellow     IN 050          20091 / 00071            30041             O.Data[2].1
   //                             IN 051          20092 / 00072            30042
   //  Door Latch Power           IN 052          20093 / 00073            30043             O.Data[2].3
   //  Safety Relay Reset         IN 053          20094 / 00074            30044             O.Data[2].4
   1: NOP();
   // Virtual Inputs
   //  These signals are sent from the PLC to the Robot. They are purely communication between the devices, so there are no physical signals attached.
   //  Name                          Robot Input     Ext. Input Signal     PLC Output
   // ---------------------------------------------------------------------------------
   //  Left Pallet Complete            IN 065             20110            O.Data[4].0
   //  Right Pallet Complete           IN 066             20111            O.Data[4].1
   //  Part In Gripper                 IN 067             20112            O.Data[4].2
   //  Gripper Extended                IN 068             20113            O.Data[4].3
   //  Gripper Retracted               IN 069             20114            O.Data[4].4
   //  Place Request Acknowledge       IN 070             20115            O.Data[4].5
   //  Check Complete Acknowledge      IN 071             20116            O.Data[4].6
   //  Pickup Error Acknowledge        IN 072             20117            O.Data[4].7
   //  Single Stack                    IN 073             20120            O.Data[5].0
   //  Quad Stack                      IN 074             20121            O.Data[5].1
   //  In Approach Acknowledge         IN 075             20122            O.Data[5].2
   //  Door Access Requested           IN 076             20123            O.Data[5].3
   //  HMI Stop                        IN 077             20124            O.Data[5].4
   //  Pick Request Acknowledge        IN 078             20125            O.Data[5].5
   //  Is Even Layer                   IN 079             20126            O.Data[5].6
   2: NOP();
   // Virtual Outputs
   //  These signals are sent from the Robot to the PLC. They are purely communication between the devices, so there are no physical signals attached.
   //  Name                   Robot Output     Ext. Ouput Signal     PLC Input
   // -----------------------------------------------------------------------------------
   //  Extend Gripper           OUT 033                             I.Data[9].0
   //  Retract Gripper          OUT 034                             I.Data[9].1
   //  Place Request            OUT 035                             I.Data[9].2
   //  Pickup Error             OUT 036                             I.Data[9].3
   //  In Approach Position     OUT 037                             I.Data[9].4
   //  Check Complete           OUT 038                             I.Data[9].5
   //  Pick Request             OUT 039                             I.Data[9].6
   3: NOP();
   // Robot Control
   //  These are intended to be physical inputs, but virtual signals from the PLC to the Robot have been mapped to the corresponding logic numbers.
   //  Name                Robot Input     Ext. Input Signal     PLC Output
   // -----------------------------------------------------------------------
   //  External Start        IN 033          20010 / 00050       O.Data[0].0
   //  External Hold         IN 034          20011 / 00051       O.Data[0].1
   //  Call Master           IN 035          20012 / 00052       O.Data[0].2
   //  Alarm Reset           IN 036          20013 / 00053       O.Data[0].3
   //  External Servo On     IN 037          20014 / 00054       O.Data[0].4
   //  Select Play Mode      IN 038          20015 / 00055       O.Data[0].5
   //  Select Teach Mode     IN 039          20016 / 00056       O.Data[0].6
   4: NOP();
   // Robot Status
   //  These are status bits that tell the PLC the state of the robot. There are no physical signals attached.
   //  Name                 Ext. Output Signal     PLC Input
   // --------------------------------------------------------
   //  Running                    30010           I.Data[8].0
   //  Servo On                   30011           I.Data[8].1
   //  Top of Master              30012           I.Data[8].2
   //  Alarm/Error Occurred       30013           I.Data[8].3
   //  Battery Alarm              30014           I.Data[8].4
   //  Remote Mode Selected       30015           I.Data[8].5
   //  Play Mode Selected         30016           I.Data[8].6
   //  Teach Mode Selected        30017           I.Data[8].7
   //  Safety Circuit Broken      30110           I.Data[4].0
   //  External E-Stop            30111           I.Data[4].1
   //  Teach Pendant E-Stop       30112           I.Data[4].2
   //  At Home Position           30122           I.Data[5].2
   5: NOP();
END_ROUTINE

ROUTINE Motoman_IO_Communication   (* ladder *)
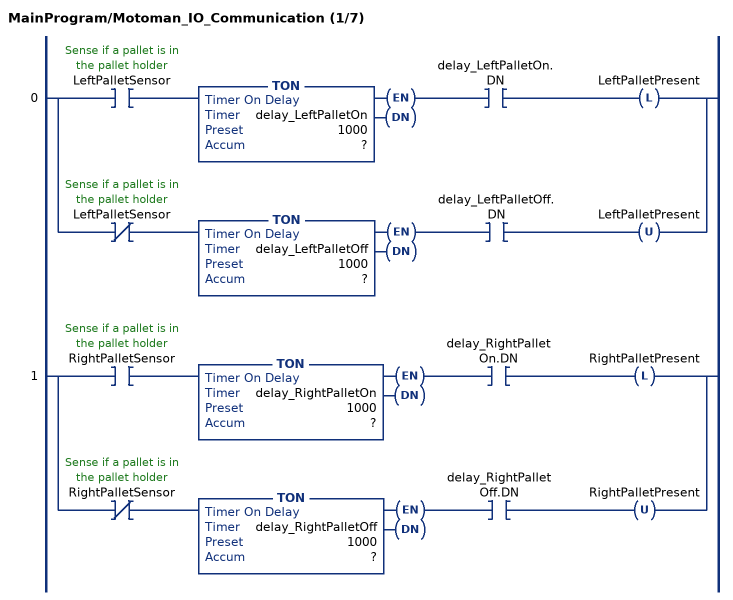
   0: [XIC(LeftPalletSensor) TON(delay_LeftPalletOn,?,?) XIC(delay_LeftPalletOn.DN) OTL(LeftPalletPresent) ,XIO(LeftPalletSensor) TON(delay_LeftPalletOff,?,?) XIC(delay_LeftPalletOff.DN) OTU(LeftPalletPresent) ];
   1: [XIC(RightPalletSensor) TON(delay_RightPalletOn,?,?) XIC(delay_RightPalletOn.DN) OTL(RightPalletPresent) ,XIO(RightPalletSensor) TON(delay_RightPalletOff,?,?) XIC(delay_RightPalletOff.DN) OTU(RightPalletPresent) ];
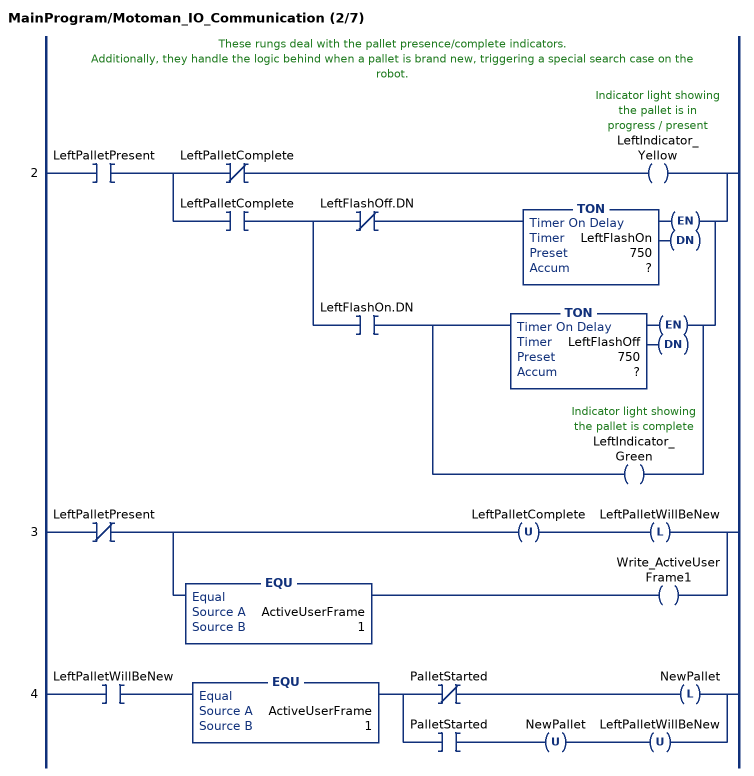
   // These rungs deal with the pallet presence/complete indicators.
   // Additionally, they handle the logic behind when a pallet is brand new, triggering a special search case on the robot.
   2: XIC(LeftPalletPresent)[XIO(LeftPalletComplete) OTE(LeftIndicator_Yellow) ,XIC(LeftPalletComplete) [XIO(LeftFlashOff.DN) TON(LeftFlashOn,?,?) ,XIC(LeftFlashOn.DN) [TON(LeftFlashOff,?,?) ,OTE(LeftIndicator_Green) ] ] ];
   3: XIO(LeftPalletPresent)[OTU(LeftPalletComplete) OTL(LeftPalletWillBeNew) ,EQU(ActiveUserFrame,1) OTE(Write_ActiveUserFrame1) ];
   4: XIC(LeftPalletWillBeNew)EQU(ActiveUserFrame,1)[XIO(PalletStarted) OTL(NewPallet) ,XIC(PalletStarted) OTU(NewPallet) OTU(LeftPalletWillBeNew) ];
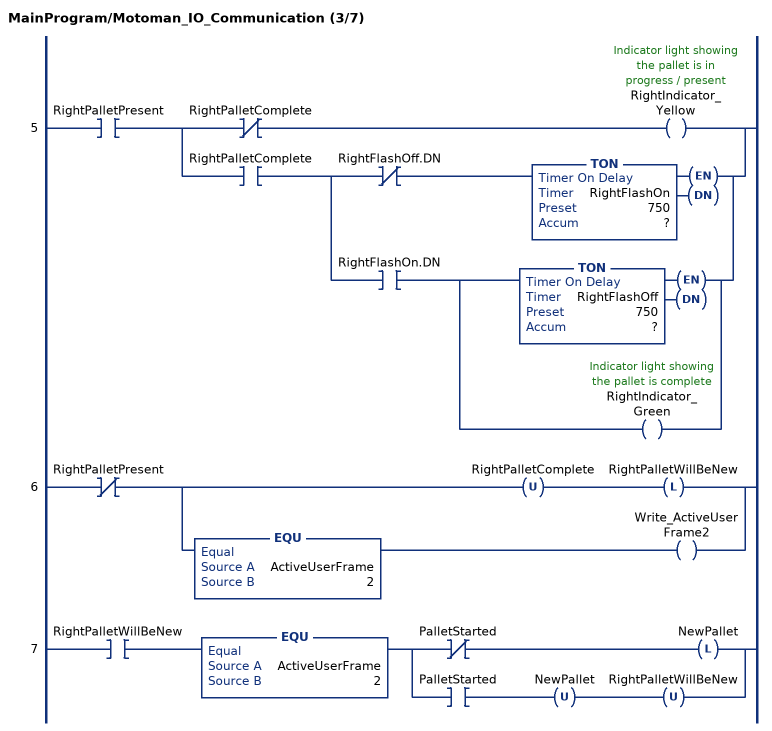
   5: XIC(RightPalletPresent)[XIO(RightPalletComplete) OTE(RightIndicator_Yellow) ,XIC(RightPalletComplete) [XIO(RightFlashOff.DN) TON(RightFlashOn,?,?) ,XIC(RightFlashOn.DN) [TON(RightFlashOff,?,?) ,OTE(RightIndicator_Green) ] ] ];
   6: XIO(RightPalletPresent)[OTU(RightPalletComplete) OTL(RightPalletWillBeNew) ,EQU(ActiveUserFrame,2) OTE(Write_ActiveUserFrame2) ];
   7: XIC(RightPalletWillBeNew)EQU(ActiveUserFrame,2)[XIO(PalletStarted) OTL(NewPallet) ,XIC(PalletStarted) OTU(NewPallet) OTU(RightPalletWillBeNew) ];
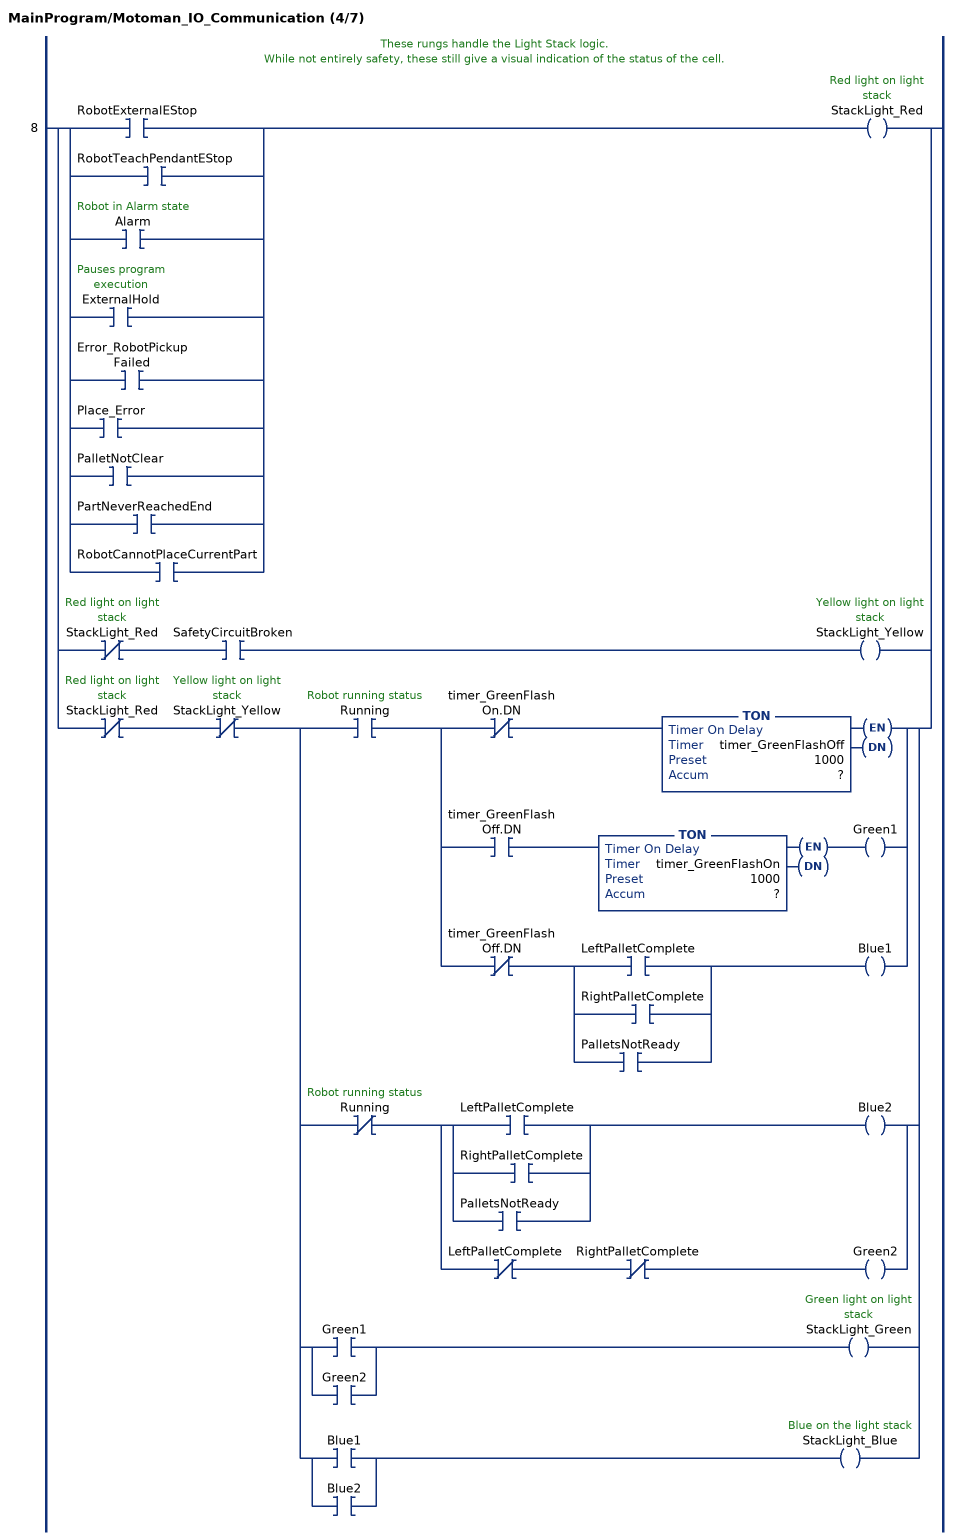
   // These rungs handle the Light Stack logic.
   // While not entirely safety, these still give a visual indication of the status of the cell.
   8: [[XIC(RobotExternalEStop) ,XIC(RobotTeachPendantEStop) ,XIC(Alarm) ,XIC(ExternalHold) ,XIC(Error_RobotPickupFailed) ,XIC(Place_Error) ,XIC(PalletNotClear) ,XIC(PartNeverReachedEnd) ,XIC(RobotCannotPlaceCurrentPart) ] OTE(StackLight_Red) ,XIO(StackLight_Red) XIC(SafetyCircuitBroken) OTE(StackLight_Yellow) ,XIO(StackLight_Red) XIO(StackLight_Yellow) [[XIC(Running) [XIO(timer_GreenFlashOn.DN) TON(timer_GreenFlashOff,?,?) ,XIC(timer_GreenFlashOff.DN) TON(timer_GreenFlashOn,?,?) OTE(Green1) ,XIO(timer_GreenFlashOff.DN) [XIC(LeftPalletComplete) ,XIC(RightPalletComplete) ,XIC(PalletsNotReady) ] OTE(Blue1) ] ,XIO(Running) [[XIC(LeftPalletComplete) ,XIC(RightPalletComplete) ,XIC(PalletsNotReady) ] OTE(Blue2) ,XIO(LeftPalletComplete) XIO(RightPalletComplete) OTE(Green2) ] ] ,[XIC(Green1) ,XIC(Green2) ] OTE(StackLight_Green) ,[XIC(Blue1) ,XIC(Blue2) ] OTE(StackLight_Blue) ] ];
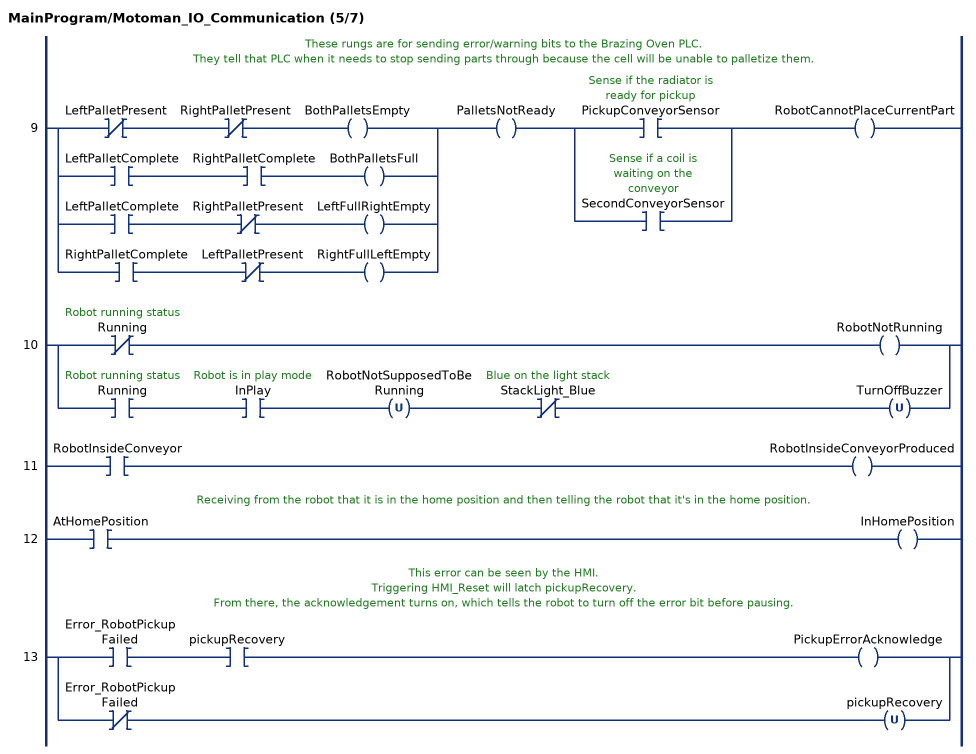
   // These rungs are for sending error/warning bits to the Brazing Oven PLC.
   // They tell that PLC when it needs to stop sending parts through because the cell will be unable to palletize them.
   9: [XIO(LeftPalletPresent) XIO(RightPalletPresent) OTE(BothPalletsEmpty) ,XIC(LeftPalletComplete) XIC(RightPalletComplete) OTE(BothPalletsFull) ,XIC(LeftPalletComplete) XIO(RightPalletPresent) OTE(LeftFullRightEmpty) ,XIC(RightPalletComplete) XIO(LeftPalletPresent) OTE(RightFullLeftEmpty) ]OTE(PalletsNotReady)[XIC(PickupConveyorSensor) ,XIC(SecondConveyorSensor) ]OTE(RobotCannotPlaceCurrentPart);
   10: [XIO(Running) OTE(RobotNotRunning) ,XIC(Running) XIC(InPlay) OTU(RobotNotSupposedToBeRunning) XIO(StackLight_Blue) OTU(TurnOffBuzzer) ];
   11: XIC(RobotInsideConveyor)OTE(RobotInsideConveyorProduced);
   // Receiving from the robot that it is in the home position and then telling the robot that it's in the home position.
   12: XIC(AtHomePosition)OTE(InHomePosition);
   // This error can be seen by the HMI.
   // Triggering HMI_Reset will latch pickupRecovery.
   // From there, the acknowledgement turns on, which tells the robot to turn off the error bit before pausing.
   13: [XIC(Error_RobotPickupFailed) XIC(pickupRecovery) OTE(PickupErrorAcknowledge) ,XIO(Error_RobotPickupFailed) OTU(pickupRecovery) ];
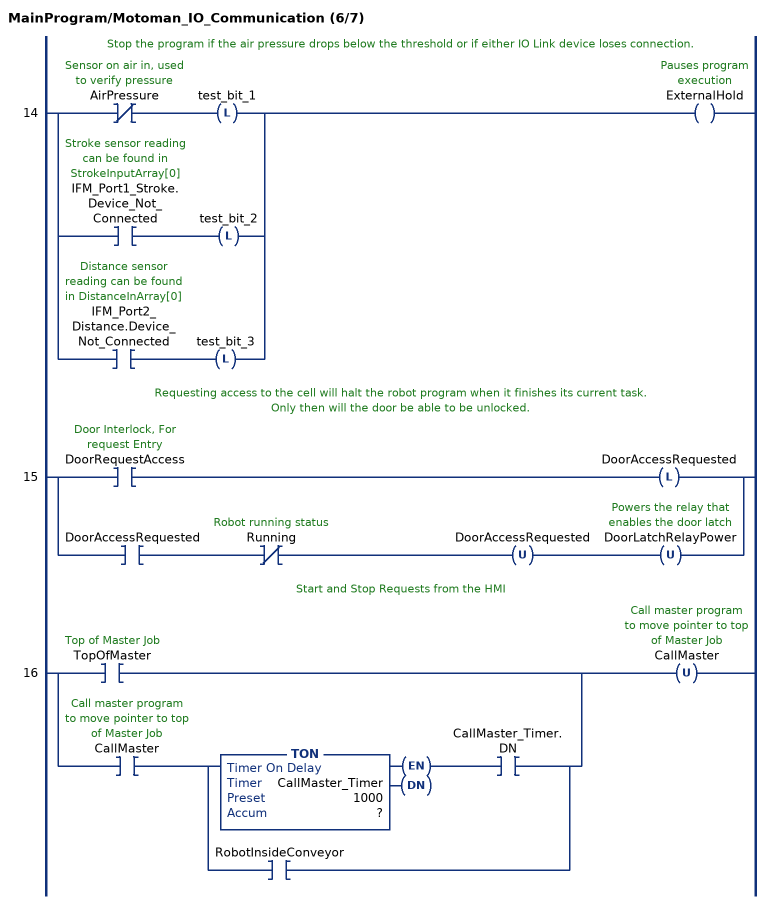
   // Stop the program if the air pressure drops below the threshold or if either IO Link device loses connection.
   14: [XIO(AirPressure) OTL(test_bit_1) ,XIC(IFM_Port1_Stroke.Device_Not_Connected) OTL(test_bit_2) ,XIC(IFM_Port2_Distance.Device_Not_Connected) OTL(test_bit_3) ]OTE(ExternalHold);
   // Requesting access to the cell will halt the robot program when it finishes its current task.
   // Only then will the door be able to be unlocked.
   15: [XIC(DoorRequestAccess) OTL(DoorAccessRequested) ,XIC(DoorAccessRequested) XIO(Running) OTU(DoorAccessRequested) OTU(DoorLatchRelayPower) ];
   // Start and Stop Requests from the HMI
   16: [XIC(TopOfMaster) ,XIC(CallMaster) [TON(CallMaster_Timer,?,?) XIC(CallMaster_Timer.DN) ,XIC(RobotInsideConveyor) ] ]OTU(CallMaster);
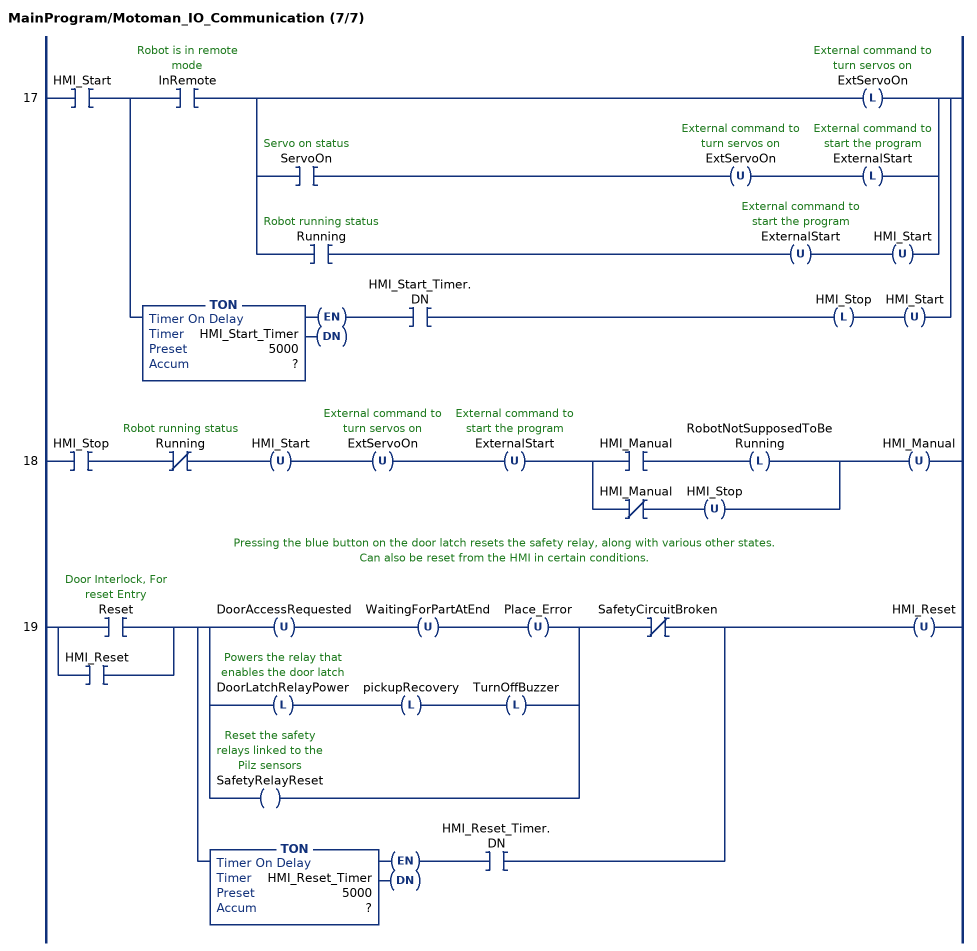
   17: XIC(HMI_Start)[XIC(InRemote) [OTL(ExtServoOn) ,XIC(ServoOn) OTU(ExtServoOn) OTL(ExternalStart) ,XIC(Running) OTU(ExternalStart) OTU(HMI_Start) ] ,TON(HMI_Start_Timer,?,?) XIC(HMI_Start_Timer.DN) OTL(HMI_Stop) OTU(HMI_Start) ];
   18: XIC(HMI_Stop)XIO(Running)OTU(HMI_Start)OTU(ExtServoOn)OTU(ExternalStart)[XIC(HMI_Manual) OTL(RobotNotSupposedToBeRunning) ,XIO(HMI_Manual) OTU(HMI_Stop) ]OTU(HMI_Manual);
   // Pressing the blue button on the door latch resets the safety relay, along with various other states.
   // Can also be reset from the HMI in certain conditions.
   19: [XIC(Reset) ,XIC(HMI_Reset) ][[OTU(DoorAccessRequested) OTU(WaitingForPartAtEnd) OTU(Place_Error) ,OTL(DoorLatchRelayPower) OTL(pickupRecovery) OTL(TurnOffBuzzer) ,OTE(SafetyRelayReset) ] XIO(SafetyCircuitBroken) ,TON(HMI_Reset_Timer,?,?) XIC(HMI_Reset_Timer.DN) ]OTU(HMI_Reset);
END_ROUTINE
